LIN {X 0,Y 343.974,Z 466.655,A -85,B 0,C 180,E1 15502.924,E2 15502.924} C_VEL
LIN {X 0,Y 341.205,Z 461.554,A -85,B 0,C 180,E1 15499.694,E2 15499.694} C_VEL
LIN {X 0,Y 339.187,Z 457.553,A -85,B 0,C 180,E1 15496.615,E2 15496.615} C_VEL
LIN {X 0,Y 338.279,Z 456.355,A -85,B 0,C 180,E1 15495.252,E2 15495.252} C_VEL
LIN {X 0,Y 336.252,Z 451.923,A -85,B 0,C 180,E1 15489.413,E2 15489.413} C_VEL
LIN {X 0,Y 335.796,Z 451.415,A -85,B 0,C 180,E1 15484.054,E2 15484.054} C_VEL
LIN {X 0,Y 336.908,Z 452.402,A -85,B 0,C 180,E1 15479.66,E2 15479.66} C_VEL
LIN {X 0,Y 340.362,Z 458.036,A -85,B 0,C 180,E1 15473.083,E2 15473.083} C_VEL
LIN {X 0,Y 342.566,Z 462.05,A -85,B 0,C 180,E1 15470.254,E2 15470.254} C_VEL
LIN {X 0,Y 343.564,Z 463.39,A -85,B 0,C 180,E1 15469.266,E2 15469.266} C_VEL
LIN {X 0,Y 346.154,Z 467.623,A -85,B 0,C 180,E1 15466.895,E2 15466.895} C_VEL
LIN {X 0,Y 352.008,Z 475.085,A -85,B 0,C 180,E1 15463.838,E2 15463.838} C_VEL
LIN {X 0,Y 358.537,Z 483.415,A -85,B 0,C 180,E1 15460.957,E2 15460.957} C_VEL
LIN {X 0,Y 366.447,Z 494.283,A -85,B 0,C 180,E1 15457.924,E2 15457.924} C_VEL
LIN {X 0,Y 375.438,Z 507.505,A -85,B 0,C 180,E1 15454.906,E2 15454.906} C_VEL
LIN {X 0,Y 384.953,Z 522.741,A -85,B 0,C 180,E1 15452.064,E2 15452.064} C_VEL
LIN {X 0,Y 386.963,Z 526.463,A -85,B 0,C 180,E1 15451.489,E2 15451.489} C_VEL
LIN {X 0,Y 374.82,Z 720.746,A -85,B 0,C 180,E1 15447.413,E2 15447.413} C_VEL
LIN {X 0,Y 369.926,Z 797.825,A -85,B 0,C 180,E1 15445.731,E2 15445.731} C_VEL
LIN {X 0,Y 367.045,Z 821.363,A -85,B 0,C 180,E1 15445.019,E2 15445.019} C_VEL
LIN {X 0,Y 363.025,Z 845.088,A -85,B 0,C 180,E1 15444.072,E2 15444.072} C_VEL
LIN {X 0,Y 358.533,Z 867.366,A -85,B 0,C 180,E1 15442.901,E2 15442.901} C_VEL
LIN {X 0,Y 353.441,Z 888.781,A -85,B 0,C 180,E1 15441.463,E2 15441.463} C_VEL
LIN {X 0,Y 347.685,Z 910.726,A -85,B 0,C 180,E1 15439.648,E2 15439.648} C_VEL
LIN {X 0,Y 341.955,Z 930.881,A -85,B 0,C 180,E1 15437.632,E2 15437.632} C_VEL
LIN {X 0,Y 335.907,Z 950.699,A -85,B 0,C 180,E1 15435.229,E2 15435.229} C_VEL
LIN {X 0,Y 329.81,Z 970.146,A -85,B 0,C 180,E1 15432.419,E2 15432.419} C_VEL
LIN {X 0,Y 324.313,Z 987.655,A -85,B 0,C 180,E1 15429.428,E2 15429.428} C_VEL
LIN {X 0,Y 319.205,Z 1004.098,A -85,B 0,C 180,E1 15426.078,E2 15426.078} C_VEL
LIN {X 0,Y 314.594,Z 1019.874,A -85,B 0,C 180,E1 15422.285,E2 15422.285} C_VEL
LIN {X 0,Y 311.178,Z 1032.9,A -85,B 0,C 180,E1 15418.605,E2 15418.605} C_VEL
LIN {X 0,Y 308.521,Z 1044.406,A -85,B 0,C 180,E1 15414.713,E2 15414.713} C_VEL
LIN {X 0,Y 306.649,Z 1054.589,A -85,B 0,C 180,E1 15410.619,E2 15410.619} C_VEL
LIN {X 0,Y 305.659,Z 1062.099,A -85,B 0,C 180,E1 15406.926,E2 15406.926} C_VEL
LIN {X 0,Y 305.155,Z 1068.715,A -85,B 0,C 180,E1 15402.874,E2 15402.874} C_VEL
LIN {X 0,Y 305.04,Z 1073.096,A -85,B 0,C 180,E1 15399.242,E2 15399.242} C_VEL
LIN {X 0,Y 305.141,Z 1075.999,A -85,B 0,C 180,E1 15395.83,E2 15395.83} C_VEL
LIN {X 0,Y 305.246,Z 1077.669,A -85,B 0,C 180,E1 15392.065,E2 15392.065} C_VEL
LIN {X 0,Y 305.248,Z 1077.813,A -85,B 0,C 180,E1 15388.874,E2 15388.874} C_VEL
LIN {X 0,Y 305.192,Z 1076.833,A -85,B 0,C 180,E1 15385.679,E2 15385.679} C_VEL
LIN {X 0,Y 305.078,Z 1074.266,A -85,B 0,C 180,E1 15381.898,E2 15381.898} C_VEL
LIN {X 0,Y 305.105,Z 1069.978,A -85,B 0,C 180,E1 15378.085,E2 15378.085} C_VEL
LIN {X 0,Y 305.427,Z 1064.526,A -85,B 0,C 180,E1 15374.428,E2 15374.428} C_VEL
LIN {X 0,Y 306.341,Z 1056.686,A -85,B 0,C 180,E1 15370.356,E2 15370.356} C_VEL
LIN {X 0,Y 307.902,Z 1047.568,A -85,B 0,C 180,E1 15366.458,E2 15366.458} C_VEL
LIN {X 0,Y 310.287,Z 1036.485,A -85,B 0,C 180,E1 15362.561,E2 15362.561} C_VEL
LIN {X 0,Y 313.609,Z 1023.525,A -85,B 0,C 180,E1 15358.689,E2 15358.689} C_VEL
LIN {X 0,Y 317.476,Z 1009.897,A -85,B 0,C 180,E1 15355.246,E2 15355.246} C_VEL
LIN {X 0,Y 322.515,Z 993.292,A -85,B 0,C 180,E1 15351.681,E2 15351.681} C_VEL
LIN {X 0,Y 327.889,Z 976.235,A -85,B 0,C 180,E1 15348.569,E2 15348.569} C_VEL
LIN {X 0,Y 333.337,Z 958.875,A -85,B 0,C 180,E1 15345.901,E2 15345.901} C_VEL
LIN {X 0,Y 339.647,Z 938.285,A -85,B 0,C 180,E1 15343.231,E2 15343.231} C_VEL
LIN {X 0,Y 345.607,Z 918.087,A -85,B 0,C 180,E1 15341.05,E2 15341.05} C_VEL
LIN {X 0,Y 351.134,Z 897.689,A -85,B 0,C 180,E1 15339.238,E2 15339.238} C_VEL
LIN {X 0,Y 356.626,Z 875.444,A -85,B 0,C 180,E1 15337.623,E2 15337.623} C_VEL
LIN {X 0,Y 361.328,Z 853.913,A -85,B 0,C 180,E1 15336.365,E2 15336.365} C_VEL
LIN {X 0,Y 365.391,Z 831.587,A -85,B 0,C 180,E1 15335.367,E2 15335.367} C_VEL
LIN {X 0,Y 368.882,Z 806.789,A -85,B 0,C 180,E1 15334.53,E2 15334.53} C_VEL
LIN {X 0,Y 370.981,Z 782.961,A -85,B 0,C 180,E1 15333.928,E2 15333.928} C_VEL
LIN {X 0,Y 383.67,Z 577.593,A -85,B 0,C 180,E1 15329.572,E2 15329.572} C_VEL
LIN {X 0,Y 386.794,Z 526.022,A -85,B 0,C 180,E1 15328.485,E2 15328.485} C_VEL
LIN {X 0,Y 378.081,Z 511.736,A -85,B 0,C 180,E1 15325.955,E2 15325.955} C_VEL
LIN {X 0,Y 370.52,Z 500.263,A -85,B 0,C 180,E1 15323.539,E2 15323.539} C_VEL
LIN {X 0,Y 361.938,Z 488.016,A -85,B 0,C 180,E1 15320.454,E2 15320.454} C_VEL
LIN {X 0,Y 354.015,Z 477.663,A -85,B 0,C 180,E1 15317.166,E2 15317.166} C_VEL
LIN {X 0,Y 349.793,Z 472.376,A -85,B 0,C 180,E1 15315.161,E2 15315.161} C_VEL
LIN {X 0,Y 345.844,Z 467.344,A -85,B 0,C 180,E1 15313.032,E2 15313.032} C_VEL
LIN {X 0,Y 342.959,Z 462.497,A -85,B 0,C 180,E1 15310.243,E2 15310.243} C_VEL
LIN {X 0,Y 340.424,Z 458.382,A -85,B 0,C 180,E1 15307.255,E2 15307.255} C_VEL
LIN {X 0,Y 339.834,Z 457.343,A -85,B 0,C 180,E1 15306.419,E2 15306.419} C_VEL
LIN {X 0,Y 336.702,Z 452.103,A -85,B 0,C 180,E1 15300.17,E2 15300.17} C_VEL
LIN {X 0,Y 335.523,Z 451.26,A -85,B 0,C 180,E1 15294.87,E2 15294.87} C_VEL
LIN {X 0,Y 336.345,Z 451.99,A -85,B 0,C 180,E1 15289.898,E2 15289.898} C_VEL
LIN {X 0,Y 339.121,Z 457.459,A -85,B 0,C 180,E1 15283.205,E2 15283.205} C_VEL
LIN {X 0,Y 341.044,Z 461.387,A -85,B 0,C 180,E1 15280.238,E2 15280.238} C_VEL
LIN {X 0,Y 341.808,Z 462.804,A -85,B 0,C 180,E1 15279.27,E2 15279.27} C_VEL
LIN {X 0,Y 344.202,Z 467.421,A -85,B 0,C 180,E1 15276.548,E2 15276.548} C_VEL
LIN {X 0,Y 348.739,Z 473.746,A -85,B 0,C 180,E1 15273.844,E2 15273.844} C_VEL
LIN {X 0,Y 351.856,Z 477.832,A -85,B 0,C 180,E1 15272.314,E2 15272.314} C_VEL
LIN {X 0,Y 358.049,Z 486.342,A -85,B 0,C 180,E1 15269.592,E2 15269.592} C_VEL
LIN {X 0,Y 364.787,Z 496.023,A -85,B 0,C 180,E1 15266.994,E2 15266.994} C_VEL
LIN {X 0,Y 372.893,Z 508.428,A -85,B 0,C 180,E1 15264.229,E2 15264.229} C_VEL
LIN {X 0,Y 381.885,Z 523.465,A -85,B 0,C 180,E1 15261.502,E2 15261.502} C_VEL
LIN {X 0,Y 381.997,Z 527.297,A -85,B 0,C 180,E1 15261.356,E2 15261.356} C_VEL
LIN {X 0,Y 370.72,Z 754.722,A -85,B 0,C 180,E1 15257.08,E2 15257.08} C_VEL
LIN {X 0,Y 368.846,Z 775.36,A -85,B 0,C 180,E1 15256.438,E2 15256.438} C_VEL
LIN {X 0,Y 366.004,Z 796.186,A -85,B 0,C 180,E1 15255.536,E2 15255.536} C_VEL
LIN {X 0,Y 362.593,Z 815.194,A -85,B 0,C 180,E1 15254.46,E2 15254.46} C_VEL
LIN {X 0,Y 358.372,Z 833.832,A -85,B 0,C 180,E1 15253.122,E2 15253.122} C_VEL
LIN {X 0,Y 353.575,Z 851.659,A -85,B 0,C 180,E1 15251.54,E2 15251.54} C_VEL
LIN {X 0,Y 348.388,Z 868.504,A -85,B 0,C 180,E1 15249.722,E2 15249.722} C_VEL
LIN {X 0,Y 342.699,Z 884.886,A -85,B 0,C 180,E1 15247.574,E2 15247.574} C_VEL
LIN {X 0,Y 336.914,Z 899.931,A -85,B 0,C 180,E1 15245.151,E2 15245.151} C_VEL
LIN {X 0,Y 331.245,Z 913.564,A -85,B 0,C 180,E1 15242.5,E2 15242.5} C_VEL
LIN {X 0,Y 325.925,Z 925.847,A -85,B 0,C 180,E1 15239.598,E2 15239.598} C_VEL
LIN {X 0,Y 320.751,Z 937.321,A -85,B 0,C 180,E1 15236.273,E2 15236.273} C_VEL
LIN {X 0,Y 316.26,Z 947.14,A -85,B 0,C 180,E1 15232.688,E2 15232.688} C_VEL
LIN {X 0,Y 312.692,Z 955.048,A -85,B 0,C 180,E1 15229.036,E2 15229.036} C_VEL
LIN {X 0,Y 309.839,Z 961.81,A -85,B 0,C 180,E1 15224.961,E2 15224.961} C_VEL
LIN {X 0,Y 308.026,Z 966.572,A -85,B 0,C 180,E1 15221.041,E2 15221.041} C_VEL
LIN {X 0,Y 306.914,Z 969.924,A -85,B 0,C 180,E1 15216.923,E2 15216.923} C_VEL
LIN {X 0,Y 306.384,Z 971.643,A -85,B 0,C 180,E1 15212.806,E2 15212.806} C_VEL
LIN {X 0,Y 306.299,Z 971.927,A -85,B 0,C 180,E1 15208.878,E2 15208.878} C_VEL
LIN {X 0,Y 306.619,Z 970.836,A -85,B 0,C 180,E1 15204.761,E2 15204.761} C_VEL
LIN {X 0,Y 307.474,Z 968.249,A -85,B 0,C 180,E1 15200.643,E2 15200.643} C_VEL
LIN {X 0,Y 309.005,Z 963.97,A -85,B 0,C 180,E1 15196.528,E2 15196.528} C_VEL
LIN {X 0,Y 311.364,Z 958.227,A -85,B 0,C 180,E1 15192.624,E2 15192.624} C_VEL
LIN {X 0,Y 314.49,Z 951.056,A -85,B 0,C 180,E1 15188.907,E2 15188.907} C_VEL
LIN {X 0,Y 314.88,Z 948.415,A -85,B 0,C 180,E1 15187.58,E2 15187.58} C_VEL
LIN {X 0,Y 313.132,Z 941.752,A -85,B 0,C 180,E1 15184.124,E2 15184.124} C_VEL
LIN {X 0,Y 313.889,Z 938.359,A -85,B 0,C 180,E1 15182.856,E2 15182.856} C_VEL
LIN {X 0,Y 319.273,Z 926.988,A -85,B 0,C 180,E1 15179.514,E2 15179.514} C_VEL
LIN {X 0,Y 324.842,Z 914.675,A -85,B 0,C 180,E1 15176.567,E2 15176.567} C_VEL
LIN {X 0,Y 331.139,Z 900.064,A -85,B 0,C 180,E1 15173.714,E2 15173.714} C_VEL
LIN {X 0,Y 336.987,Z 885.362,A -85,B 0,C 180,E1 15171.349,E2 15171.349} C_VEL
LIN {X 0,Y 342.841,Z 869.118,A -85,B 0,C 180,E1 15169.211,E2 15169.211} C_VEL
LIN {X 0,Y 348.074,Z 852.672,A -85,B 0,C 180,E1 15167.43,E2 15167.43} C_VEL
LIN {X 0,Y 353.045,Z 834.833,A -85,B 0,C 180,E1 15165.837,E2 15165.837} C_VEL
LIN {X 0,Y 357.415,Z 816.203,A -85,B 0,C 180,E1 15164.491,E2 15164.491} C_VEL
LIN {X 0,Y 361.075,Z 796.506,A -85,B 0,C 180,E1 15163.373,E2 15163.373} C_VEL
LIN {X 0,Y 364.016,Z 775.499,A -85,B 0,C 180,E1 15162.468,E2 15162.468} C_VEL
LIN {X 0,Y 365.927,Z 754.887,A -85,B 0,C 180,E1 15161.83,E2 15161.83} C_VEL
LIN {X 0,Y 377.655,Z 527.845,A -85,B 0,C 180,E1 15157.513,E2 15157.513} C_VEL
LIN {X 0,Y 369.147,Z 513.555,A -85,B 0,C 180,E1 15154.809,E2 15154.809} C_VEL
LIN {X 0,Y 361.207,Z 501.26,A -85,B 0,C 180,E1 15151.965,E2 15151.965} C_VEL
LIN {X 0,Y 354.549,Z 491.6,A -85,B 0,C 180,E1 15149.248,E2 15149.248} C_VEL
LIN {X 0,Y 348.202,Z 482.708,A -85,B 0,C 180,E1 15146.245,E2 15146.245} C_VEL
LIN {X 0,Y 341.714,Z 474.041,A -85,B 0,C 180,E1 15142.539,E2 15142.539} C_VEL
LIN {X 0,Y 338.064,Z 469.215,A -85,B 0,C 180,E1 15139.975,E2 15139.975} C_VEL
LIN {X 0,Y 335.758,Z 465.827,A -85,B 0,C 180,E1 15137.326,E2 15137.326} C_VEL
LIN {X 0,Y 335.009,Z 463.83,A -85,B 0,C 180,E1 15135.76,E2 15135.76} C_VEL
LIN {X 0,Y 332.7,Z 459.081,A -85,B 0,C 180,E1 15129.34,E2 15129.34} C_VEL
LIN {X 0,Y 332.274,Z 458.602,A -85,B 0,C 180,E1 15123.969,E2 15123.969} C_VEL
LIN {X 0,Y 333.405,Z 459.621,A -85,B 0,C 180,E1 15119.657,E2 15119.657} C_VEL
LIN {X 0,Y 336.734,Z 465.24,A -85,B 0,C 180,E1 15113.179,E2 15113.179} C_VEL
LIN {X 0,Y 338.642,Z 468.549,A -85,B 0,C 180,E1 15110.998,E2 15110.998} C_VEL
LIN {X 0,Y 340.885,Z 470.946,A -85,B 0,C 180,E1 15109.437,E2 15109.437} C_VEL
LIN {X 0,Y 345.367,Z 476.472,A -85,B 0,C 180,E1 15106.694,E2 15106.694} C_VEL
LIN {X 0,Y 350.089,Z 482.514,A -85,B 0,C 180,E1 15104.215,E2 15104.215} C_VEL
LIN {X 0,Y 356.404,Z 490.785,A -85,B 0,C 180,E1 15101.349,E2 15101.349} C_VEL
LIN {X 0,Y 363.89,Z 501.241,A -85,B 0,C 180,E1 15098.396,E2 15098.396} C_VEL
LIN {X 0,Y 372.816,Z 514.664,A -85,B 0,C 180,E1 15095.311,E2 15095.311} C_VEL
LIN {X 0,Y 381.781,Z 529.373,A -85,B 0,C 180,E1 15092.553,E2 15092.553} C_VEL
LIN {X 0,Y 382.259,Z 530.611,A -85,B 0,C 180,E1 15092.4,E2 15092.4} C_VEL
LIN {X 0,Y 369.496,Z 728.067,A -85,B 0,C 180,E1 15088.238,E2 15088.238} C_VEL
LIN {X 0,Y 364.921,Z 797.295,A -85,B 0,C 180,E1 15086.716,E2 15086.716} C_VEL
LIN {X 0,Y 361.961,Z 820.778,A -85,B 0,C 180,E1 15086.002,E2 15086.002} C_VEL
LIN {X 0,Y 357.789,Z 844.591,A -85,B 0,C 180,E1 15085.049,E2 15085.049} C_VEL
LIN {X 0,Y 353.133,Z 866.83,A -85,B 0,C 180,E1 15083.875,E2 15083.875} C_VEL
LIN {X 0,Y 347.716,Z 888.76,A -85,B 0,C 180,E1 15082.392,E2 15082.392} C_VEL
LIN {X 0,Y 341.748,Z 910.507,A -85,B 0,C 180,E1 15080.57,E2 15080.57} C_VEL
LIN {X 0,Y 335.713,Z 930.832,A -85,B 0,C 180,E1 15078.503,E2 15078.503} C_VEL
LIN {X 0,Y 329.57,Z 950.06,A -85,B 0,C 180,E1 15076.133,E2 15076.133} C_VEL
LIN {X 0,Y 323.088,Z 969.683,A -85,B 0,C 180,E1 15073.246,E2 15073.246} C_VEL
LIN {X 0,Y 317.223,Z 987.432,A -85,B 0,C 180,E1 15070.134,E2 15070.134} C_VEL
LIN {X 0,Y 312.017,Z 1003.337,A -85,B 0,C 180,E1 15066.816,E2 15066.816} C_VEL
LIN {X 0,Y 307.367,Z 1018.332,A -85,B 0,C 180,E1 15063.128,E2 15063.128} C_VEL
LIN {X 0,Y 303.597,Z 1031.821,A -85,B 0,C 180,E1 15059.222,E2 15059.222} C_VEL
LIN {X 0,Y 300.754,Z 1043.422,A -85,B 0,C 180,E1 15055.185,E2 15055.185} C_VEL
LIN {X 0,Y 298.775,Z 1053.528,A -85,B 0,C 180,E1 15050.982,E2 15050.982} C_VEL
LIN {X 0,Y 297.731,Z 1061.003,A -85,B 0,C 180,E1 15047.189,E2 15047.189} C_VEL
LIN {X 0,Y 297.219,Z 1067.547,A -85,B 0,C 180,E1 15043.026,E2 15043.026} C_VEL
LIN {X 0,Y 297.115,Z 1071.696,A -85,B 0,C 180,E1 15039.491,E2 15039.491} C_VEL
LIN {X 0,Y 297.245,Z 1074.62,A -85,B 0,C 180,E1 15035.985,E2 15035.985} C_VEL
LIN {X 0,Y 297.358,Z 1076.302,A -85,B 0,C 180,E1 15032.12,E2 15032.12} C_VEL
LIN {X 0,Y 297.365,Z 1076.447,A -85,B 0,C 180,E1 15028.844,E2 15028.844} C_VEL
LIN {X 0,Y 297.294,Z 1075.458,A -85,B 0,C 180,E1 15025.563,E2 15025.563} C_VEL
LIN {X 0,Y 297.164,Z 1073.048,A -85,B 0,C 180,E1 15021.876,E2 15021.876} C_VEL
LIN {X 0,Y 297.174,Z 1068.811,A -85,B 0,C 180,E1 15017.959,E2 15017.959} C_VEL
LIN {X 0,Y 297.499,Z 1063.392,A -85,B 0,C 180,E1 15014.203,E2 15014.203} C_VEL
LIN {X 0,Y 298.443,Z 1055.623,A -85,B 0,C 180,E1 15010.018,E2 15010.018} C_VEL
LIN {X 0,Y 299.989,Z 1047.02,A -85,B 0,C 180,E1 15006.216,E2 15006.216} C_VEL
LIN {X 0,Y 302.462,Z 1036.135,A -85,B 0,C 180,E1 15002.218,E2 15002.218} C_VEL
LIN {X 0,Y 305.92,Z 1023.385,A -85,B 0,C 180,E1 14998.25,E2 14998.25} C_VEL
LIN {X 0,Y 310.195,Z 1009.083,A -85,B 0,C 180,E1 14994.535,E2 14994.535} C_VEL
LIN {X 0,Y 315.486,Z 992.578,A -85,B 0,C 180,E1 14990.899,E2 14990.899} C_VEL
LIN {X 0,Y 321.139,Z 975.638,A -85,B 0,C 180,E1 14987.738,E2 14987.738} C_VEL
LIN {X 0,Y 327.07,Z 957.6,A -85,B 0,C 180,E1 14984.923,E2 14984.923} C_VEL
LIN {X 0,Y 333.629,Z 937.172,A -85,B 0,C 180,E1 14982.248,E2 14982.248} C_VEL
LIN {X 0,Y 339.766,Z 917.287,A -85,B 0,C 180,E1 14980.081,E2 14980.081} C_VEL
LIN {X 0,Y 345.491,Z 896.992,A -85,B 0,C 180,E1 14978.266,E2 14978.266} C_VEL
LIN {X 0,Y 351.284,Z 874.352,A -85,B 0,C 180,E1 14976.615,E2 14976.615} C_VEL
LIN {X 0,Y 356.178,Z 852.663,A -85,B 0,C 180,E1 14975.35,E2 14975.35} C_VEL
LIN {X 0,Y 360.379,Z 830.197,A -85,B 0,C 180,E1 14974.352,E2 14974.352} C_VEL
LIN {X 0,Y 363.929,Z 805.476,A -85,B 0,C 180,E1 14973.525,E2 14973.525} C_VEL
LIN {X 0,Y 366.084,Z 781.261,A -85,B 0,C 180,E1 14972.916,E2 14972.916} C_VEL
LIN {X 0,Y 379.142,Z 577.108,A -85,B 0,C 180,E1 14968.57,E2 14968.57} C_VEL
LIN {X 0,Y 382.085,Z 530.038,A -85,B 0,C 180,E1 14967.571,E2 14967.571} C_VEL
LIN {X 0,Y 374.108,Z 516.865,A -85,B 0,C 180,E1 14965.147,E2 14965.147} C_VEL
LIN {X 0,Y 367.26,Z 506.362,A -85,B 0,C 180,E1 14962.869,E2 14962.869} C_VEL
LIN {X 0,Y 359.461,Z 494.995,A -85,B 0,C 180,E1 14959.964,E2 14959.964} C_VEL
LIN {X 0,Y 351.97,Z 484.981,A -85,B 0,C 180,E1 14956.758,E2 14956.758} C_VEL
LIN {X 0,Y 347.835,Z 479.71,A -85,B 0,C 180,E1 14954.737,E2 14954.737} C_VEL
LIN {X 0,Y 343.952,Z 474.731,A -85,B 0,C 180,E1 14952.592,E2 14952.592} C_VEL
LIN {X 0,Y 339.747,Z 469.644,A -85,B 0,C 180,E1 14949.913,E2 14949.913} C_VEL
LIN {X 0,Y 336.992,Z 466.115,A -85,B 0,C 180,E1 14947.501,E2 14947.501} C_VEL
LIN {X 0,Y 336.247,Z 464.471,A -85,B 0,C 180,E1 14946.316,E2 14946.316} C_VEL
LIN {X 0,Y 333.205,Z 459.312,A -85,B 0,C 180,E1 14940.171,E2 14940.171} C_VEL
LIN {X 0,Y 331.998,Z 458.438,A -85,B 0,C 180,E1 14934.989,E2 14934.989} C_VEL
LIN {X 0,Y 332.745,Z 459.126,A -85,B 0,C 180,E1 14929.963,E2 14929.963} C_VEL
LIN {X 0,Y 335.313,Z 464.463,A -85,B 0,C 180,E1 14923.365,E2 14923.365} C_VEL
LIN {X 0,Y 337.249,Z 468.357,A -85,B 0,C 180,E1 14920.426,E2 14920.426} C_VEL
LIN {X 0,Y 338.525,Z 470.119,A -85,B 0,C 180,E1 14919.422,E2 14919.422} C_VEL
LIN {X 0,Y 342.714,Z 475.552,A -85,B 0,C 180,E1 14916.623,E2 14916.623} C_VEL
LIN {X 0,Y 348.932,Z 483.649,A -85,B 0,C 180,E1 14913.217,E2 14913.217} C_VEL
LIN {X 0,Y 356.118,Z 493.943,A -85,B 0,C 180,E1 14909.922,E2 14909.922} C_VEL
LIN {X 0,Y 362.767,Z 503.721,A -85,B 0,C 180,E1 14907.301,E2 14907.301} C_VEL
LIN {X 0,Y 370.116,Z 515.249,A -85,B 0,C 180,E1 14904.729,E2 14904.729} C_VEL
LIN {X 0,Y 377.635,Z 528.076,A -85,B 0,C 180,E1 14902.361,E2 14902.361} C_VEL
LIN {X 0,Y 365.808,Z 755.43,A -85,B 0,C 180,E1 14898.056,E2 14898.056} C_VEL
LIN {X 0,Y 363.855,Z 776.124,A -85,B 0,C 180,E1 14897.409,E2 14897.409} C_VEL
LIN {X 0,Y 360.866,Z 797.225,A -85,B 0,C 180,E1 14896.489,E2 14896.489} C_VEL
LIN {X 0,Y 357.174,Z 816.9,A -85,B 0,C 180,E1 14895.36,E2 14895.36} C_VEL
LIN {X 0,Y 352.734,Z 835.787,A -85,B 0,C 180,E1 14893.986,E2 14893.986} C_VEL
LIN {X 0,Y 347.747,Z 853.498,A -85,B 0,C 180,E1 14892.385,E2 14892.385} C_VEL
LIN {X 0,Y 341.876,Z 871.62,A -85,B 0,C 180,E1 14890.377,E2 14890.377} C_VEL
LIN {X 0,Y 336.095,Z 887.515,A -85,B 0,C 180,E1 14888.228,E2 14888.228} C_VEL
LIN {X 0,Y 330.137,Z 902.402,A -85,B 0,C 180,E1 14885.77,E2 14885.77} C_VEL
LIN {X 0,Y 324.277,Z 915.819,A -85,B 0,C 180,E1 14883.076,E2 14883.076} C_VEL
LIN {X 0,Y 318.428,Z 928.63,A -85,B 0,C 180,E1 14879.929,E2 14879.929} C_VEL
LIN {X 0,Y 313.346,Z 939.384,A -85,B 0,C 180,E1 14876.688,E2 14876.688} C_VEL
LIN {X 0,Y 308.76,Z 949.009,A -85,B 0,C 180,E1 14873.069,E2 14873.069} C_VEL
LIN {X 0,Y 304.958,Z 957.012,A -85,B 0,C 180,E1 14869.219,E2 14869.219} C_VEL
LIN {X 0,Y 302.19,Z 963.193,A -85,B 0,C 180,E1 14865.349,E2 14865.349} C_VEL
LIN {X 0,Y 300.19,Z 968.121,A -85,B 0,C 180,E1 14861.139,E2 14861.139} C_VEL
LIN {X 0,Y 299.077,Z 971.293,A -85,B 0,C 180,E1 14857.106,E2 14857.106} C_VEL
LIN {X 0,Y 298.507,Z 973.01,A -85,B 0,C 180,E1 14852.88,E2 14852.88} C_VEL
LIN {X 0,Y 298.418,Z 973.292,A -85,B 0,C 180,E1 14848.848,E2 14848.848} C_VEL
LIN {X 0,Y 298.761,Z 972.203,A -85,B 0,C 180,E1 14844.623,E2 14844.623} C_VEL
LIN {X 0,Y 299.674,Z 969.621,A -85,B 0,C 180,E1 14840.397,E2 14840.397} C_VEL
LIN {X 0,Y 301.307,Z 965.347,A -85,B 0,C 180,E1 14836.177,E2 14836.177} C_VEL
LIN {X 0,Y 303.804,Z 959.612,A -85,B 0,C 180,E1 14832.177,E2 14832.177} C_VEL
LIN {X 0,Y 307.259,Z 952.126,A -85,B 0,C 180,E1 14828.224,E2 14828.224} C_VEL
LIN {X 0,Y 311.57,Z 943.154,A -85,B 0,C 180,E1 14824.531,E2 14824.531} C_VEL
LIN {X 0,Y 313.889,Z 938.359,A -85,B 0,C 180,E1 14822.856,E2 14822.856} C_VEL
LIN {X 0,Y 314.744,Z 934.836,A -85,B 0,C 180,E1 14821.61,E2 14821.61} C_VEL
LIN {X 0,Y 314.325,Z 926.159,A -85,B 0,C 180,E1 14818.307,E2 14818.307} C_VEL
LIN {X 0,Y 315.576,Z 921.965,A -85,B 0,C 180,E1 14817.129,E2 14817.129} C_VEL
LIN {X 0,Y 321.754,Z 908.546,A -85,B 0,C 180,E1 14814.201,E2 14814.201} C_VEL
LIN {X 0,Y 328.22,Z 893.534,A -85,B 0,C 180,E1 14811.528,E2 14811.528} C_VEL
LIN {X 0,Y 334.217,Z 878.324,A -85,B 0,C 180,E1 14809.294,E2 14809.294} C_VEL
LIN {X 0,Y 340.217,Z 861.159,A -85,B 0,C 180,E1 14807.243,E2 14807.243} C_VEL
LIN {X 0,Y 345.516,Z 843.84,A -85,B 0,C 180,E1 14805.548,E2 14805.548} C_VEL
LIN {X 0,Y 350.34,Z 825.554,A -85,B 0,C 180,E1 14804.087,E2 14804.087} C_VEL
LIN {X 0,Y 354.296,Z 807.283,A -85,B 0,C 180,E1 14802.917,E2 14802.917} C_VEL
LIN {X 0,Y 357.665,Z 787.369,A -85,B 0,C 180,E1 14801.919,E2 14801.919} C_VEL
LIN {X 0,Y 360.171,Z 766.869,A -85,B 0,C 180,E1 14801.148,E2 14801.148} C_VEL
LIN {X 0,Y 361.729,Z 745.715,A -85,B 0,C 180,E1 14800.6,E2 14800.6} C_VEL
LIN {X 0,Y 373.246,Z 531.923,A -85,B 0,C 180,E1 14796.552,E2 14796.552} C_VEL
LIN {X 0,Y 364.866,Z 517.88,A -85,B 0,C 180,E1 14793.753,E2 14793.753} C_VEL
LIN {X 0,Y 357.885,Z 506.971,A -85,B 0,C 180,E1 14791.122,E2 14791.122} C_VEL
LIN {X 0,Y 351.891,Z 498.044,A -85,B 0,C 180,E1 14788.56,E2 14788.56} C_VEL
LIN {X 0,Y 346.048,Z 489.737,A -85,B 0,C 180,E1 14785.684,E2 14785.684} C_VEL
LIN {X 0,Y 340.123,Z 481.605,A -85,B 0,C 180,E1 14782.179,E2 14782.179} C_VEL
LIN {X 0,Y 335.951,Z 476.14,A -85,B 0,C 180,E1 14779.11,E2 14779.11} C_VEL
LIN {X 0,Y 332.24,Z 471.267,A -85,B 0,C 180,E1 14775.536,E2 14775.536} C_VEL
LIN {X 0,Y 329.308,Z 466.828,A -85,B 0,C 180,E1 14770.32,E2 14770.32} C_VEL
LIN {X 0,Y 328.869,Z 465.945,A -85,B 0,C 180,E1 14767.864,E2 14767.864} C_VEL
LIN {X 0,Y 329.092,Z 466.025,A -85,B 0,C 180,E1 14762.264,E2 14762.264} C_VEL
LIN {X 0,Y 329.974,Z 467.019,A -85,B 0,C 180,E1 14759.397,E2 14759.397} C_VEL
LIN {X 0,Y 334.712,Z 472.907,A -85,B 0,C 180,E1 14753.396,E2 14753.396} C_VEL
LIN {X 0,Y 339.413,Z 478.686,A -85,B 0,C 180,E1 14749.712,E2 14749.712} C_VEL
LIN {X 0,Y 343.638,Z 483.995,A -85,B 0,C 180,E1 14747.054,E2 14747.054} C_VEL
LIN {X 0,Y 348.185,Z 489.944,A -85,B 0,C 180,E1 14744.596,E2 14744.596} C_VEL
LIN {X 0,Y 354.208,Z 498.011,A -85,B 0,C 180,E1 14741.783,E2 14741.783} C_VEL
LIN {X 0,Y 361.449,Z 508.343,A -85,B 0,C 180,E1 14738.839,E2 14738.839} C_VEL
LIN {X 0,Y 370.105,Z 521.665,A -85,B 0,C 180,E1 14735.756,E2 14735.756} C_VEL
LIN {X 0,Y 377.68,Z 534.326,A -85,B 0,C 180,E1 14733.341,E2 14733.341} C_VEL
LIN {X 0,Y 364.39,Z 733.159,A -85,B 0,C 180,E1 14729.135,E2 14729.135} C_VEL
LIN {X 0,Y 360.038,Z 796.661,A -85,B 0,C 180,E1 14727.73,E2 14727.73} C_VEL
LIN {X 0,Y 356.981,Z 820.227,A -85,B 0,C 180,E1 14727.012,E2 14727.012} C_VEL
LIN {X 0,Y 352.754,Z 843.661,A -85,B 0,C 180,E1 14726.075,E2 14726.075} C_VEL
LIN {X 0,Y 348.076,Z 865.368,A -85,B 0,C 180,E1 14724.936,E2 14724.936} C_VEL
LIN {X 0,Y 342.643,Z 886.645,A -85,B 0,C 180,E1 14723.508,E2 14723.508} C_VEL
LIN {X 0,Y 336.42,Z 908.571,A -85,B 0,C 180,E1 14721.686,E2 14721.686} C_VEL
LIN {X 0,Y 330.087,Z 929.157,A -85,B 0,C 180,E1 14719.593,E2 14719.593} C_VEL
LIN {X 0,Y 323.86,Z 947.813,A -85,B 0,C 180,E1 14717.289,E2 14717.289} C_VEL
LIN {X 0,Y 317.12,Z 967.302,A -85,B 0,C 180,E1 14714.424,E2 14714.424} C_VEL
LIN {X 0,Y 311.046,Z 984.829,A -85,B 0,C 180,E1 14711.345,E2 14711.345} C_VEL
LIN {X 0,Y 305.33,Z 1001.246,A -85,B 0,C 180,E1 14707.89,E2 14707.89} C_VEL
LIN {X 0,Y 300.153,Z 1016.986,A -85,B 0,C 180,E1 14703.958,E2 14703.958} C_VEL
LIN {X 0,Y 296.141,Z 1030.423,A -85,B 0,C 180,E1 14699.98,E2 14699.98} C_VEL
LIN {X 0,Y 293.127,Z 1041.904,A -85,B 0,C 180,E1 14695.888,E2 14695.888} C_VEL
LIN {X 0,Y 290.913,Z 1052.47,A -85,B 0,C 180,E1 14691.366,E2 14691.366} C_VEL
LIN {X 0,Y 289.809,Z 1059.911,A -85,B 0,C 180,E1 14687.467,E2 14687.467} C_VEL
LIN {X 0,Y 289.284,Z 1066.38,A -85,B 0,C 180,E1 14683.186,E2 14683.186} C_VEL
LIN {X 0,Y 289.192,Z 1070.494,A -85,B 0,C 180,E1 14679.553,E2 14679.553} C_VEL
LIN {X 0,Y 289.34,Z 1073.514,A -85,B 0,C 180,E1 14675.751,E2 14675.751} C_VEL
LIN {X 0,Y 289.479,Z 1074.966,A -85,B 0,C 180,E1 14671.979,E2 14671.979} C_VEL
LIN {X 0,Y 289.485,Z 1075.054,A -85,B 0,C 180,E1 14668.615,E2 14668.615} C_VEL
LIN {X 0,Y 289.372,Z 1073.908,A -85,B 0,C 180,E1 14665.044,E2 14665.044} C_VEL
LIN {X 0,Y 289.209,Z 1071.08,A -85,B 0,C 180,E1 14661.05,E2 14661.05} C_VEL
LIN {X 0,Y 289.255,Z 1067.139,A -85,B 0,C 180,E1 14657.422,E2 14657.422} C_VEL
LIN {X 0,Y 289.662,Z 1061.325,A -85,B 0,C 180,E1 14653.351,E2 14653.351} C_VEL
LIN {X 0,Y 290.687,Z 1053.721,A -85,B 0,C 180,E1 14649.25,E2 14649.25} C_VEL
LIN {X 0,Y 292.514,Z 1044.553,A -85,B 0,C 180,E1 14645.138,E2 14645.138} C_VEL
LIN {X 0,Y 295.281,Z 1033.396,A -85,B 0,C 180,E1 14641.039,E2 14641.039} C_VEL
LIN {X 0,Y 299.086,Z 1020.351,A -85,B 0,C 180,E1 14636.981,E2 14636.981} C_VEL
LIN {X 0,Y 303.494,Z 1006.686,A -85,B 0,C 180,E1 14633.394,E2 14633.394} C_VEL
LIN {X 0,Y 309.027,Z 990.385,A -85,B 0,C 180,E1 14629.78,E2 14629.78} C_VEL
LIN {X 0,Y 314.921,Z 973.655,A -85,B 0,C 180,E1 14626.64,E2 14626.64} C_VEL
LIN {X 0,Y 321.089,Z 955.805,A -85,B 0,C 180,E1 14623.83,E2 14623.83} C_VEL
LIN {X 0,Y 327.753,Z 935.968,A -85,B 0,C 180,E1 14621.218,E2 14621.218} C_VEL
LIN {X 0,Y 334.159,Z 916.054,A -85,B 0,C 180,E1 14619.038,E2 14619.038} C_VEL
LIN {X 0,Y 339.898,Z 896.488,A -85,B 0,C 180,E1 14617.277,E2 14617.277} C_VEL
LIN {X 0,Y 345.772,Z 874.449,A -85,B 0,C 180,E1 14615.652,E2 14615.652} C_VEL
LIN {X 0,Y 350.647,Z 853.646,A -85,B 0,C 180,E1 14614.425,E2 14614.425} C_VEL
LIN {X 0,Y 355.083,Z 831.103,A -85,B 0,C 180,E1 14613.402,E2 14613.402} C_VEL
LIN {X 0,Y 358.691,Z 807.631,A -85,B 0,C 180,E1 14612.591,E2 14612.591} C_VEL
LIN {X 0,Y 360.959,Z 784.51,A -85,B 0,C 180,E1 14611.989,E2 14611.989} C_VEL
LIN {X 0,Y 374.374,Z 582.053,A -85,B 0,C 180,E1 14607.658,E2 14607.658} C_VEL
LIN {X 0,Y 377.495,Z 534.077,A -85,B 0,C 180,E1 14606.637,E2 14606.637} C_VEL
LIN {X 0,Y 368.44,Z 519.057,A -85,B 0,C 180,E1 14603.722,E2 14603.722} C_VEL
LIN {X 0,Y 359.603,Z 505.746,A -85,B 0,C 180,E1 14600.507,E2 14600.507} C_VEL
LIN {X 0,Y 352.593,Z 495.932,A -85,B 0,C 180,E1 14597.577,E2 14597.577} C_VEL
LIN {X 0,Y 346.508,Z 487.717,A -85,B 0,C 180,E1 14594.624,E2 14594.624} C_VEL
LIN {X 0,Y 342.11,Z 482.12,A -85,B 0,C 180,E1 14592.147,E2 14592.147} C_VEL
LIN {X 0,Y 338.147,Z 477.2,A -85,B 0,C 180,E1 14589.531,E2 14589.531} C_VEL
LIN {X 0,Y 334.065,Z 472.129,A -85,B 0,C 180,E1 14586.185,E2 14586.185} C_VEL
LIN {X 0,Y 329.765,Z 466.613,A -85,B 0,C 180,E1 14580.347,E2 14580.347} C_VEL
LIN {X 0,Y 328.508,Z 465.626,A -85,B 0,C 180,E1 14575.286,E2 14575.286} C_VEL
LIN {X 0,Y 329.143,Z 466.26,A -85,B 0,C 180,E1 14570.028,E2 14570.028} C_VEL
LIN {X 0,Y 330.569,Z 469.617,A -85,B 0,C 180,E1 14566.149,E2 14566.149} C_VEL
LIN {X 0,Y 332.75,Z 471.94,A -85,B 0,C 180,E1 14563.593,E2 14563.593} C_VEL
LIN {X 0,Y 336.09,Z 476.274,A -85,B 0,C 180,E1 14560.537,E2 14560.537} C_VEL
LIN {X 0,Y 341.18,Z 483.221,A -85,B 0,C 180,E1 14556.927,E2 14556.927} C_VEL
LIN {X 0,Y 347.061,Z 491.081,A -85,B 0,C 180,E1 14553.616,E2 14553.616} C_VEL
LIN {X 0,Y 353.848,Z 500.995,A -85,B 0,C 180,E1 14550.41,E2 14550.41} C_VEL
LIN {X 0,Y 360.951,Z 511.682,A -85,B 0,C 180,E1 14547.54,E2 14547.54} C_VEL
LIN {X 0,Y 368.648,Z 524.259,A -85,B 0,C 180,E1 14544.805,E2 14544.805} C_VEL
LIN {X 0,Y 373.199,Z 532.134,A -85,B 0,C 180,E1 14543.328,E2 14543.328} C_VEL
LIN {X 0,Y 361.005,Z 756.112,A -85,B 0,C 180,E1 14539.059,E2 14539.059} C_VEL
LIN {X 0,Y 358.97,Z 776.874,A -85,B 0,C 180,E1 14538.407,E2 14538.407} C_VEL
LIN {X 0,Y 355.829,Z 798.251,A -85,B 0,C 180,E1 14537.469,E2 14537.469} C_VEL
LIN {X 0,Y 352.126,Z 817.386,A -85,B 0,C 180,E1 14536.37,E2 14536.37} C_VEL
LIN {X 0,Y 347.66,Z 835.802,A -85,B 0,C 180,E1 14535.031,E2 14535.031} C_VEL
LIN {X 0,Y 342.566,Z 853.498,A -85,B 0,C 180,E1 14533.442,E2 14533.442} C_VEL
LIN {X 0,Y 336.877,Z 870.721,A -85,B 0,C 180,E1 14531.557,E2 14531.557} C_VEL
LIN {X 0,Y 330.831,Z 886.924,A -85,B 0,C 180,E1 14529.396,E2 14529.396} C_VEL
LIN {X 0,Y 324.575,Z 902.026,A -85,B 0,C 180,E1 14526.921,E2 14526.921} C_VEL
LIN {X 0,Y 318.424,Z 915.724,A -85,B 0,C 180,E1 14524.199,E2 14524.199} C_VEL
LIN {X 0,Y 312.608,Z 928.077,A -85,B 0,C 180,E1 14521.208,E2 14521.208} C_VEL
LIN {X 0,Y 307.18,Z 939.03,A -85,B 0,C 180,E1 14517.951,E2 14517.951} C_VEL
LIN {X 0,Y 302.375,Z 948.569,A -85,B 0,C 180,E1 14514.415,E2 14514.415} C_VEL
LIN {X 0,Y 298.096,Z 957.117,A -85,B 0,C 180,E1 14510.416,E2 14510.416} C_VEL
LIN {X 0,Y 294.933,Z 963.787,A -85,B 0,C 180,E1 14506.343,E2 14506.343} C_VEL
LIN {X 0,Y 292.658,Z 968.973,A -85,B 0,C 180,E1 14502.029,E2 14502.029} C_VEL
LIN {X 0,Y 291.327,Z 972.399,A -85,B 0,C 180,E1 14497.692,E2 14497.692} C_VEL
LIN {X 0,Y 290.671,Z 974.207,A -85,B 0,C 180,E1 14493.55,E2 14493.55} C_VEL
LIN {X 0,Y 290.528,Z 974.696,A -85,B 0,C 180,E1 14489.211,E2 14489.211} C_VEL
LIN {X 0,Y 290.827,Z 973.848,A -85,B 0,C 180,E1 14485.069,E2 14485.069} C_VEL
LIN {X 0,Y 291.696,Z 971.4,A -85,B 0,C 180,E1 14480.729,E2 14480.729} C_VEL
LIN {X 0,Y 293.318,Z 967.376,A -85,B 0,C 180,E1 14476.396,E2 14476.396} C_VEL
LIN {X 0,Y 295.976,Z 961.614,A -85,B 0,C 180,E1 14472.096,E2 14472.096} C_VEL
LIN {X 0,Y 299.519,Z 954.337,A -85,B 0,C 180,E1 14468.045,E2 14468.045} C_VEL
LIN {X 0,Y 303.952,Z 945.585,A -85,B 0,C 180,E1 14464.264,E2 14464.264} C_VEL
LIN {X 0,Y 309.075,Z 935.299,A -85,B 0,C 180,E1 14460.759,E2 14460.759} C_VEL
LIN {X 0,Y 314.787,Z 923.595,A -85,B 0,C 180,E1 14457.534,E2 14457.534} C_VEL
LIN {X 0,Y 315.576,Z 921.965,A -85,B 0,C 180,E1 14457.129,E2 14457.129} C_VEL
LIN {X 0,Y 316.903,Z 917.709,A -85,B 0,C 180,E1 14455.976,E2 14455.976} C_VEL
LIN {X 0,Y 317.547,Z 906.996,A -85,B 0,C 180,E1 14452.904,E2 14452.904} C_VEL
LIN {X 0,Y 319.035,Z 902.075,A -85,B 0,C 180,E1 14451.858,E2 14451.858} C_VEL
LIN {X 0,Y 325.552,Z 886.801,A -85,B 0,C 180,E1 14449.374,E2 14449.374} C_VEL
LIN {X 0,Y 331.862,Z 870.461,A -85,B 0,C 180,E1 14447.203,E2 14447.203} C_VEL
LIN {X 0,Y 337.733,Z 853.06,A -85,B 0,C 180,E1 14445.322,E2 14445.322} C_VEL
LIN {X 0,Y 343.209,Z 834.236,A -85,B 0,C 180,E1 14443.666,E2 14443.666} C_VEL
LIN {X 0,Y 347.882,Z 815.095,A -85,B 0,C 180,E1 14442.316,E2 14442.316} C_VEL
LIN {X 0,Y 351.673,Z 795.599,A -85,B 0,C 180,E1 14441.235,E2 14441.235} C_VEL
LIN {X 0,Y 354.566,Z 775.461,A -85,B 0,C 180,E1 14440.39,E2 14440.39} C_VEL
LIN {X 0,Y 356.608,Z 753.633,A -85,B 0,C 180,E1 14439.734,E2 14439.734} C_VEL
LIN {X 0,Y 368.894,Z 536.076,A -85,B 0,C 180,E1 14435.558,E2 14435.558} C_VEL
LIN {X 0,Y 361.606,Z 523.659,A -85,B 0,C 180,E1 14433.006,E2 14433.006} C_VEL
LIN {X 0,Y 354.739,Z 512.766,A -85,B 0,C 180,E1 14430.3,E2 14430.3} C_VEL
LIN {X 0,Y 347.912,Z 502.382,A -85,B 0,C 180,E1 14427.191,E2 14427.191} C_VEL
LIN {X 0,Y 343.494,Z 496.172,A -85,B 0,C 180,E1 14424.874,E2 14424.874} C_VEL
LIN {X 0,Y 338.218,Z 488.823,A -85,B 0,C 180,E1 14421.596,E2 14421.596} C_VEL
LIN {X 0,Y 334.61,Z 483.857,A -85,B 0,C 180,E1 14418.828,E2 14418.828} C_VEL
LIN {X 0,Y 331.146,Z 479.157,A -85,B 0,C 180,E1 14415.409,E2 14415.409} C_VEL
LIN {X 0,Y 327.571,Z 474.054,A -85,B 0,C 180,E1 14409.133,E2 14409.133} C_VEL
LIN {X 0,Y 327.192,Z 473.669,A -85,B 0,C 180,E1 14403.68,E2 14403.68} C_VEL
LIN {X 0,Y 328.571,Z 474.67,A -85,B 0,C 180,E1 14399.826,E2 14399.826} C_VEL
LIN {X 0,Y 333.424,Z 480.721,A -85,B 0,C 180,E1 14393.63,E2 14393.63} C_VEL
LIN {X 0,Y 337.89,Z 486.327,A -85,B 0,C 180,E1 14390.032,E2 14390.032} C_VEL
LIN {X 0,Y 341.989,Z 491.618,A -85,B 0,C 180,E1 14387.377,E2 14387.377} C_VEL
LIN {X 0,Y 346.301,Z 497.372,A -85,B 0,C 180,E1 14384.982,E2 14384.982} C_VEL
LIN {X 0,Y 352.115,Z 505.367,A -85,B 0,C 180,E1 14382.184,E2 14382.184} C_VEL
LIN {X 0,Y 359.119,Z 515.586,A -85,B 0,C 180,E1 14379.251,E2 14379.251} C_VEL
LIN {X 0,Y 367.415,Z 528.694,A -85,B 0,C 180,E1 14376.207,E2 14376.207} C_VEL
LIN {X 0,Y 373.174,Z 538.512,A -85,B 0,C 180,E1 14374.297,E2 14374.297} C_VEL
LIN {X 0,Y 359.217,Z 740.845,A -85,B 0,C 180,E1 14370.003,E2 14370.003} C_VEL
LIN {X 0,Y 355.257,Z 796.184,A -85,B 0,C 180,E1 14368.768,E2 14368.768} C_VEL
LIN {X 0,Y 352.122,Z 819.667,A -85,B 0,C 180,E1 14368.05,E2 14368.05} C_VEL
LIN {X 0,Y 347.718,Z 843.315,A -85,B 0,C 180,E1 14367.103,E2 14367.103} C_VEL
LIN {X 0,Y 342.77,Z 865.362,A -85,B 0,C 180,E1 14365.938,E2 14365.938} C_VEL
LIN {X 0,Y 337.135,Z 886.641,A -85,B 0,C 180,E1 14364.499,E2 14364.499} C_VEL
LIN {X 0,Y 330.694,Z 908.372,A -85,B 0,C 180,E1 14362.673,E2 14362.673} C_VEL
LIN {X 0,Y 324.186,Z 928.638,A -85,B 0,C 180,E1 14360.588,E2 14360.588} C_VEL
LIN {X 0,Y 317.655,Z 947.372,A -85,B 0,C 180,E1 14358.244,E2 14358.244} C_VEL
LIN {X 0,Y 310.634,Z 966.732,A -85,B 0,C 180,E1 14355.345,E2 14355.345} C_VEL
LIN {X 0,Y 304.268,Z 984.162,A -85,B 0,C 180,E1 14352.223,E2 14352.223} C_VEL
LIN {X 0,Y 298.421,Z 1000.105,A -85,B 0,C 180,E1 14348.796,E2 14348.796} C_VEL
LIN {X 0,Y 292.911,Z 1015.911,A -85,B 0,C 180,E1 14344.755,E2 14344.755} C_VEL
LIN {X 0,Y 288.778,Z 1028.883,A -85,B 0,C 180,E1 14340.826,E2 14340.826} C_VEL
LIN {X 0,Y 285.534,Z 1040.389,A -85,B 0,C 180,E1 14336.63,E2 14336.63} C_VEL
LIN {X 0,Y 283.144,Z 1050.992,A -85,B 0,C 180,E1 14331.982,E2 14331.982} C_VEL
LIN {X 0,Y 281.942,Z 1058.456,A -85,B 0,C 180,E1 14327.971,E2 14327.971} C_VEL
LIN {X 0,Y 281.354,Z 1064.957,A -85,B 0,C 180,E1 14323.565,E2 14323.565} C_VEL
LIN {X 0,Y 281.27,Z 1069.095,A -85,B 0,C 180,E1 14319.825,E2 14319.825} C_VEL
LIN {X 0,Y 281.442,Z 1072.152,A -85,B 0,C 180,E1 14315.889,E2 14315.889} C_VEL
LIN {X 0,Y 281.59,Z 1073.599,A -85,B 0,C 180,E1 14312.035,E2 14312.035} C_VEL
LIN {X 0,Y 281.599,Z 1073.716,A -85,B 0,C 180,E1 14308.779,E2 14308.779} C_VEL
LIN {X 0,Y 281.495,Z 1072.71,A -85,B 0,C 180,E1 14305.314,E2 14305.314} C_VEL
LIN {X 0,Y 281.307,Z 1070.262,A -85,B 0,C 180,E1 14301.415,E2 14301.415} C_VEL
LIN {X 0,Y 281.32,Z 1065.973,A -85,B 0,C 180,E1 14297.27,E2 14297.27} C_VEL
LIN {X 0,Y 281.704,Z 1060.505,A -85,B 0,C 180,E1 14293.292,E2 14293.292} C_VEL
LIN {X 0,Y 282.818,Z 1052.663,A -85,B 0,C 180,E1 14288.862,E2 14288.862} C_VEL
LIN {X 0,Y 284.634,Z 1044.014,A -85,B 0,C 180,E1 14284.846,E2 14284.846} C_VEL
LIN {X 0,Y 287.507,Z 1033.054,A -85,B 0,C 180,E1 14280.636,E2 14280.636} C_VEL
LIN {X 0,Y 291.247,Z 1020.937,A -85,B 0,C 180,E1 14276.682,E2 14276.682} C_VEL
LIN {X 0,Y 296.059,Z 1006.678,A -85,B 0,C 180,E1 14272.805,E2 14272.805} C_VEL
LIN {X 0,Y 302.005,Z 990.121,A -85,B 0,C 180,E1 14269.011,E2 14269.011} C_VEL
LIN {X 0,Y 308.229,Z 973.343,A -85,B 0,C 180,E1 14265.778,E2 14265.778} C_VEL
LIN {X 0,Y 314.922,Z 954.883,A -85,B 0,C 180,E1 14262.826,E2 14262.826} C_VEL
LIN {X 0,Y 321.925,Z 934.98,A -85,B 0,C 180,E1 14260.177,E2 14260.177} C_VEL
LIN {X 0,Y 328.574,Z 915.128,A -85,B 0,C 180,E1 14257.987,E2 14257.987} C_VEL
LIN {X 0,Y 334.777,Z 894.722,A -85,B 0,C 180,E1 14256.148,E2 14256.148} C_VEL
LIN {X 0,Y 340.946,Z 872.193,A -85,B 0,C 180,E1 14254.506,E2 14254.506} C_VEL
LIN {X 0,Y 346.138,Z 850.592,A -85,B 0,C 180,E1 14253.253,E2 14253.253} C_VEL
LIN {X 0,Y 350.679,Z 827.668,A -85,B 0,C 180,E1 14252.248,E2 14252.248} C_VEL
LIN {X 0,Y 354.298,Z 803.536,A -85,B 0,C 180,E1 14251.451,E2 14251.451} C_VEL
LIN {X 0,Y 356.581,Z 778.954,A -85,B 0,C 180,E1 14250.835,E2 14250.835} C_VEL
LIN {X 0,Y 370.583,Z 574.243,A -85,B 0,C 180,E1 14246.454,E2 14246.454} C_VEL
LIN {X 0,Y 373.022,Z 538.281,A -85,B 0,C 180,E1 14245.693,E2 14245.693} C_VEL
LIN {X 0,Y 365.059,Z 524.976,A -85,B 0,C 180,E1 14243.015,E2 14243.015} C_VEL
LIN {X 0,Y 357.035,Z 512.575,A -85,B 0,C 180,E1 14239.977,E2 14239.977} C_VEL
LIN {X 0,Y 350.281,Z 502.914,A -85,B 0,C 180,E1 14237.055,E2 14237.055} C_VEL
LIN {X 0,Y 344.43,Z 494.89,A -85,B 0,C 180,E1 14234.113,E2 14234.113} C_VEL
LIN {X 0,Y 340.422,Z 489.639,A -85,B 0,C 180,E1 14231.778,E2 14231.778} C_VEL
LIN {X 0,Y 336.562,Z 484.752,A -85,B 0,C 180,E1 14229.145,E2 14229.145} C_VEL
LIN {X 0,Y 332.695,Z 479.849,A -85,B 0,C 180,E1 14225.864,E2 14225.864} C_VEL
LIN {X 0,Y 328.262,Z 474.337,A -85,B 0,C 180,E1 14219.999,E2 14219.999} C_VEL
LIN {X 0,Y 326.757,Z 473.438,A -85,B 0,C 180,E1 14214.556,E2 14214.556} C_VEL
LIN {X 0,Y 327.603,Z 474.17,A -85,B 0,C 180,E1 14209.981,E2 14209.981} C_VEL
LIN {X 0,Y 331.563,Z 479.808,A -85,B 0,C 180,E1 14203.802,E2 14203.802} C_VEL
LIN {X 0,Y 335.353,Z 484.908,A -85,B 0,C 180,E1 14200.311,E2 14200.311} C_VEL
LIN {X 0,Y 339.664,Z 490.917,A -85,B 0,C 180,E1 14197.226,E2 14197.226} C_VEL
LIN {X 0,Y 345.133,Z 498.383,A -85,B 0,C 180,E1 14194.058,E2 14194.058} C_VEL
LIN {X 0,Y 351.775,Z 508.314,A -85,B 0,C 180,E1 14190.826,E2 14190.826} C_VEL
LIN {X 0,Y 358.952,Z 519.39,A -85,B 0,C 180,E1 14187.857,E2 14187.857} C_VEL
LIN {X 0,Y 366.975,Z 532.768,A -85,B 0,C 180,E1 14184.955,E2 14184.955} C_VEL
LIN {X 0,Y 368.856,Z 536.423,A -85,B 0,C 180,E1 14184.313,E2 14184.313} C_VEL
LIN {X 0,Y 356.321,Z 756.684,A -85,B 0,C 180,E1 14180.091,E2 14180.091} C_VEL
LIN {X 0,Y 354.213,Z 777.483,A -85,B 0,C 180,E1 14179.436,E2 14179.436} C_VEL
LIN {X 0,Y 351.031,Z 798.546,A -85,B 0,C 180,E1 14178.514,E2 14178.514} C_VEL
LIN {X 0,Y 347.195,Z 817.852,A -85,B 0,C 180,E1 14177.409,E2 14177.409} C_VEL
LIN {X 0,Y 342.537,Z 836.452,A -85,B 0,C 180,E1 14176.056,E2 14176.056} C_VEL
LIN {X 0,Y 337.143,Z 854.608,A -85,B 0,C 180,E1 14174.42,E2 14174.42} C_VEL
LIN {X 0,Y 331.297,Z 871.716,A -85,B 0,C 180,E1 14172.535,E2 14172.535} C_VEL
LIN {X 0,Y 325.077,Z 887.819,A -85,B 0,C 180,E1 14170.374,E2 14170.374} C_VEL
LIN {X 0,Y 318.734,Z 902.597,A -85,B 0,C 180,E1 14167.941,E2 14167.941} C_VEL
LIN {X 0,Y 312.319,Z 916.405,A -85,B 0,C 180,E1 14165.188,E2 14165.188} C_VEL
LIN {X 0,Y 306.218,Z 928.865,A -85,B 0,C 180,E1 14162.156,E2 14162.156} C_VEL
LIN {X 0,Y 300.214,Z 940.454,A -85,B 0,C 180,E1 14158.659,E2 14158.659} C_VEL
LIN {X 0,Y 295.18,Z 949.975,A -85,B 0,C 180,E1 14155.05,E2 14155.05} C_VEL
LIN {X 0,Y 290.679,Z 958.508,A -85,B 0,C 180,E1 14150.961,E2 14150.961} C_VEL
LIN {X 0,Y 287.338,Z 965.166,A -85,B 0,C 180,E1 14146.787,E2 14146.787} C_VEL
LIN {X 0,Y 285.008,Z 970.16,A -85,B 0,C 180,E1 14142.563,E2 14142.563} C_VEL
LIN {X 0,Y 283.546,Z 973.634,A -85,B 0,C 180,E1 14138.109,E2 14138.109} C_VEL
LIN {X 0,Y 282.799,Z 975.573,A -85,B 0,C 180,E1 14133.649,E2 14133.649} C_VEL
LIN {X 0,Y 282.646,Z 976.061,A -85,B 0,C 180,E1 14129.189,E2 14129.189} C_VEL
LIN {X 0,Y 282.965,Z 975.215,A -85,B 0,C 180,E1 14124.932,E2 14124.932} C_VEL
LIN {X 0,Y 283.902,Z 972.752,A -85,B 0,C 180,E1 14120.444,E2 14120.444} C_VEL
LIN {X 0,Y 285.625,Z 968.753,A -85,B 0,C 180,E1 14116.022,E2 14116.022} C_VEL
LIN {X 0,Y 288.439,Z 962.999,A -85,B 0,C 180,E1 14111.612,E2 14111.612} C_VEL
LIN {X 0,Y 292.181,Z 955.733,A -85,B 0,C 180,E1 14107.463,E2 14107.463} C_VEL
LIN {X 0,Y 296.833,Z 946.986,A -85,B 0,C 180,E1 14103.6,E2 14103.6} C_VEL
LIN {X 0,Y 302.198,Z 936.715,A -85,B 0,C 180,E1 14100.026,E2 14100.026} C_VEL
LIN {X 0,Y 308.154,Z 925.039,A -85,B 0,C 180,E1 14096.746,E2 14096.746} C_VEL
LIN {X 0,Y 314.515,Z 911.952,A -85,B 0,C 180,E1 14093.75,E2 14093.75} C_VEL
LIN {X 0,Y 319.035,Z 902.075,A -85,B 0,C 180,E1 14091.858,E2 14091.858} C_VEL
LIN {X 0,Y 320.611,Z 897.039,A -85,B 0,C 180,E1 14090.832,E2 14090.832} C_VEL
LIN {X 0,Y 321.928,Z 884.542,A -85,B 0,C 180,E1 14088.031,E2 14088.031} C_VEL
LIN {X 0,Y 323.506,Z 878.903,A -85,B 0,C 180,E1 14087.132,E2 14087.132} C_VEL
LIN {X 0,Y 329.927,Z 861.7,A -85,B 0,C 180,E1 14085.08,E2 14085.08} C_VEL
LIN {X 0,Y 335.608,Z 844.028,A -85,B 0,C 180,E1 14083.369,E2 14083.369} C_VEL
LIN {X 0,Y 340.934,Z 824.583,A -85,B 0,C 180,E1 14081.848,E2 14081.848} C_VEL
LIN {X 0,Y 345.264,Z 805.306,A -85,B 0,C 180,E1 14080.647,E2 14080.647} C_VEL
LIN {X 0,Y 348.749,Z 784.994,A -85,B 0,C 180,E1 14079.673,E2 14079.673} C_VEL
LIN {X 0,Y 351.223,Z 764.196,A -85,B 0,C 180,E1 14078.94,E2 14078.94} C_VEL
LIN {X 0,Y 353.023,Z 737.894,A -85,B 0,C 180,E1 14078.329,E2 14078.329} C_VEL
LIN {X 0,Y 364.746,Z 540.389,A -85,B 0,C 180,E1 14074.572,E2 14074.572} C_VEL
LIN {X 0,Y 357.55,Z 527.944,A -85,B 0,C 180,E1 14071.906,E2 14071.906} C_VEL
LIN {X 0,Y 350.545,Z 516.763,A -85,B 0,C 180,E1 14068.959,E2 14068.959} C_VEL
LIN {X 0,Y 344.627,Z 507.837,A -85,B 0,C 180,E1 14066.075,E2 14066.075} C_VEL
LIN {X 0,Y 340.342,Z 501.476,A -85,B 0,C 180,E1 14063.642,E2 14063.642} C_VEL
LIN {X 0,Y 336.342,Z 496.009,A -85,B 0,C 180,E1 14061,E2 14061} C_VEL
LIN {X 0,Y 333.172,Z 491.47,A -85,B 0,C 180,E1 14058.458,E2 14058.458} C_VEL
LIN {X 0,Y 329.898,Z 486.924,A -85,B 0,C 180,E1 14055.109,E2 14055.109} C_VEL
LIN {X 0,Y 326.56,Z 481.959,A -85,B 0,C 180,E1 14048.984,E2 14048.984} C_VEL
LIN {X 0,Y 326.212,Z 481.609,A -85,B 0,C 180,E1 14043.691,E2 14043.691} C_VEL
LIN {X 0,Y 327.58,Z 482.658,A -85,B 0,C 180,E1 14039.826,E2 14039.826} C_VEL
LIN {X 0,Y 332.059,Z 488.382,A -85,B 0,C 180,E1 14033.951,E2 14033.951} C_VEL
LIN {X 0,Y 336.407,Z 494.012,A -85,B 0,C 180,E1 14030.333,E2 14030.333} C_VEL
LIN {X 0,Y 340.353,Z 499.237,A -85,B 0,C 180,E1 14027.703,E2 14027.703} C_VEL
LIN {X 0,Y 344.58,Z 505.016,A -85,B 0,C 180,E1 14025.292,E2 14025.292} C_VEL
LIN {X 0,Y 350.113,Z 512.847,A -85,B 0,C 180,E1 14022.551,E2 14022.551} C_VEL
LIN {X 0,Y 356.812,Z 522.825,A -85,B 0,C 180,E1 14019.668,E2 14019.668} C_VEL
LIN {X 0,Y 364.856,Z 535.89,A -85,B 0,C 180,E1 14016.63,E2 14016.63} C_VEL
LIN {X 0,Y 368.766,Z 542.826,A -85,B 0,C 180,E1 14015.273,E2 14015.273} C_VEL
LIN {X 0,Y 354.289,Z 746.122,A -85,B 0,C 180,E1 14010.948,E2 14010.948} C_VEL
LIN {X 0,Y 350.603,Z 795.634,A -85,B 0,C 180,E1 14009.836,E2 14009.836} C_VEL
LIN {X 0,Y 347.394,Z 819.046,A -85,B 0,C 180,E1 14009.12,E2 14009.12} C_VEL
LIN {X 0,Y 342.96,Z 842.241,A -85,B 0,C 180,E1 14008.194,E2 14008.194} C_VEL
LIN {X 0,Y 338.173,Z 863.108,A -85,B 0,C 180,E1 14007.108,E2 14007.108} C_VEL
LIN {X 0,Y 332.25,Z 884.847,A -85,B 0,C 180,E1 14005.655,E2 14005.655} C_VEL
LIN {X 0,Y 325.355,Z 907.318,A -85,B 0,C 180,E1 14003.775,E2 14003.775} C_VEL
LIN {X 0,Y 318.587,Z 927.562,A -85,B 0,C 180,E1 14001.685,E2 14001.685} C_VEL
LIN {X 0,Y 311.542,Z 946.94,A -85,B 0,C 180,E1 13999.237,E2 13999.237} C_VEL
LIN {X 0,Y 304.237,Z 966.169,A -85,B 0,C 180,E1 13996.305,E2 13996.305} C_VEL
LIN {X 0,Y 297.708,Z 983.121,A -85,B 0,C 180,E1 13993.215,E2 13993.215} C_VEL
LIN {X 0,Y 291.443,Z 999.363,A -85,B 0,C 180,E1 13989.652,E2 13989.652} C_VEL
LIN {X 0,Y 285.899,Z 1014.344,A -85,B 0,C 180,E1 13985.736,E2 13985.736} C_VEL
LIN {X 0,Y 281.473,Z 1027.341,A -85,B 0,C 180,E1 13981.718,E2 13981.718} C_VEL
LIN {X 0,Y 277.903,Z 1039.168,A -85,B 0,C 180,E1 13977.295,E2 13977.295} C_VEL
LIN {X 0,Y 275.306,Z 1049.938,A -85,B 0,C 180,E1 13972.417,E2 13972.417} C_VEL
LIN {X 0,Y 273.983,Z 1057.731,A -85,B 0,C 180,E1 13968.071,E2 13968.071} C_VEL
LIN {X 0,Y 273.407,Z 1064.049,A -85,B 0,C 180,E1 13963.536,E2 13963.536} C_VEL
LIN {X 0,Y 273.348,Z 1068.092,A -85,B 0,C 180,E1 13959.687,E2 13959.687} C_VEL
LIN {X 0,Y 273.548,Z 1070.98,A -85,B 0,C 180,E1 13955.664,E2 13955.664} C_VEL
LIN {X 0,Y 273.712,Z 1072.264,A -85,B 0,C 180,E1 13951.884,E2 13951.884} C_VEL
LIN {X 0,Y 273.718,Z 1072.322,A -85,B 0,C 180,E1 13948.535,E2 13948.535} C_VEL
LIN {X 0,Y 273.578,Z 1071.246,A -85,B 0,C 180,E1 13944.968,E2 13944.968} C_VEL
LIN {X 0,Y 273.362,Z 1068.674,A -85,B 0,C 180,E1 13940.949,E2 13940.949} C_VEL
LIN {X 0,Y 273.393,Z 1064.553,A -85,B 0,C 180,E1 13936.894,E2 13936.894} C_VEL
LIN {X 0,Y 273.847,Z 1058.747,A -85,B 0,C 180,E1 13932.579,E2 13932.579} C_VEL
LIN {X 0,Y 275.131,Z 1050.765,A -85,B 0,C 180,E1 13928.018,E2 13928.018} C_VEL
LIN {X 0,Y 277.28,Z 1041.537,A -85,B 0,C 180,E1 13923.67,E2 13923.67} C_VEL
LIN {X 0,Y 280.487,Z 1030.323,A -85,B 0,C 180,E1 13919.352,E2 13919.352} C_VEL
LIN {X 0,Y 285.121,Z 1016.479,A -85,B 0,C 180,E1 13914.892,E2 13914.892} C_VEL
LIN {X 0,Y 290.483,Z 1001.9,A -85,B 0,C 180,E1 13910.957,E2 13910.957} C_VEL
LIN {X 0,Y 296.629,Z 985.771,A -85,B 0,C 180,E1 13907.349,E2 13907.349} C_VEL
LIN {X 0,Y 303.578,Z 967.752,A -85,B 0,C 180,E1 13903.974,E2 13903.974} C_VEL
LIN {X 0,Y 310.59,Z 949.469,A -85,B 0,C 180,E1 13901.123,E2 13901.123} C_VEL
LIN {X 0,Y 317.276,Z 931.022,A -85,B 0,C 180,E1 13898.742,E2 13898.742} C_VEL
LIN {X 0,Y 324.506,Z 909.738,A -85,B 0,C 180,E1 13896.468,E2 13896.468} C_VEL
LIN {X 0,Y 330.834,Z 889.6,A -85,B 0,C 180,E1 13894.709,E2 13894.709} C_VEL
LIN {X 0,Y 336.58,Z 868.781,A -85,B 0,C 180,E1 13893.254,E2 13893.254} C_VEL
LIN {X 0,Y 342.286,Z 844.946,A -85,B 0,C 180,E1 13891.941,E2 13891.941} C_VEL
LIN {X 0,Y 346.81,Z 822.215,A -85,B 0,C 180,E1 13890.997,E2 13890.997} C_VEL
LIN {X 0,Y 350.12,Z 798.845,A -85,B 0,C 180,E1 13890.266,E2 13890.266} C_VEL
LIN {X 0,Y 352.784,Z 766.633,A -85,B 0,C 180,E1 13889.508,E2 13889.508} C_VEL
LIN {X 0,Y 367.519,Z 558.555,A -85,B 0,C 180,E1 13885.063,E2 13885.063} C_VEL
LIN {X 0,Y 368.564,Z 542.315,A -85,B 0,C 180,E1 13884.694,E2 13884.694} C_VEL
LIN {X 0,Y 361.15,Z 529.939,A -85,B 0,C 180,E1 13882.075,E2 13882.075} C_VEL
LIN {X 0,Y 354.404,Z 519.27,A -85,B 0,C 180,E1 13879.402,E2 13879.402} C_VEL
LIN {X 0,Y 347.516,Z 509.201,A -85,B 0,C 180,E1 13876.291,E2 13876.291} C_VEL
LIN {X 0,Y 342.381,Z 502.054,A -85,B 0,C 180,E1 13873.596,E2 13873.596} C_VEL
LIN {X 0,Y 338.623,Z 497.018,A -85,B 0,C 180,E1 13871.323,E2 13871.323} C_VEL
LIN {X 0,Y 335.105,Z 492.417,A -85,B 0,C 180,E1 13868.839,E2 13868.839} C_VEL
LIN {X 0,Y 331.336,Z 487.568,A -85,B 0,C 180,E1 13865.541,E2 13865.541} C_VEL
LIN {X 0,Y 327.187,Z 482.212,A -85,B 0,C 180,E1 13859.824,E2 13859.824} C_VEL
LIN {X 0,Y 325.787,Z 481.373,A -85,B 0,C 180,E1 13854.187,E2 13854.187} C_VEL
LIN {X 0,Y 326.633,Z 482.189,A -85,B 0,C 180,E1 13849.951,E2 13849.951} C_VEL
LIN {X 0,Y 330.299,Z 487.525,A -85,B 0,C 180,E1 13844.1,E2 13844.1} C_VEL
LIN {X 0,Y 333.992,Z 492.668,A -85,B 0,C 180,E1 13840.591,E2 13840.591} C_VEL
LIN {X 0,Y 338.089,Z 498.505,A -85,B 0,C 180,E1 13837.573,E2 13837.573} C_VEL
LIN {X 0,Y 343.37,Z 505.93,A -85,B 0,C 180,E1 13834.425,E2 13834.425} C_VEL
LIN {X 0,Y 349.554,Z 515.366,A -85,B 0,C 180,E1 13831.325,E2 13831.325} C_VEL
LIN {X 0,Y 356.578,Z 526.475,A -85,B 0,C 180,E1 13828.328,E2 13828.328} C_VEL
LIN {X 0,Y 364.14,Z 539.4,A -85,B 0,C 180,E1 13825.505,E2 13825.505} C_VEL
LIN {X 0,Y 364.618,Z 540.676,A -85,B 0,C 180,E1 13825.322,E2 13825.322} C_VEL
LIN {X 0,Y 351.749,Z 757.342,A -85,B 0,C 180,E1 13821.148,E2 13821.148} C_VEL
LIN {X 0,Y 349.557,Z 778.219,A -85,B 0,C 180,E1 13820.489,E2 13820.489} C_VEL
LIN {X 0,Y 346.216,Z 799.559,A -85,B 0,C 180,E1 13819.551,E2 13819.551} C_VEL
LIN {X 0,Y 342.176,Z 819.133,A -85,B 0,C 180,E1 13818.422,E2 13818.422} C_VEL
LIN {X 0,Y 337.354,Z 837.748,A -85,B 0,C 180,E1 13817.06,E2 13817.06} C_VEL
LIN {X 0,Y 331.841,Z 855.66,A -85,B 0,C 180,E1 13815.434,E2 13815.434} C_VEL
LIN {X 0,Y 325.817,Z 872.706,A -85,B 0,C 180,E1 13813.547,E2 13813.547} C_VEL
LIN {X 0,Y 319.324,Z 888.944,A -85,B 0,C 180,E1 13811.352,E2 13811.352} C_VEL
LIN {X 0,Y 313,Z 903.158,A -85,B 0,C 180,E1 13808.999,E2 13808.999} C_VEL
LIN {X 0,Y 305.91,Z 917.87,A -85,B 0,C 180,E1 13806.039,E2 13806.039} C_VEL
LIN {X 0,Y 299.557,Z 930.294,A -85,B 0,C 180,E1 13802.961,E2 13802.961} C_VEL
LIN {X 0,Y 293.296,Z 941.876,A -85,B 0,C 180,E1 13799.4,E2 13799.4} C_VEL
LIN {X 0,Y 288.023,Z 951.375,A -85,B 0,C 180,E1 13795.718,E2 13795.718} C_VEL
LIN {X 0,Y 283.29,Z 959.897,A -85,B 0,C 180,E1 13791.535,E2 13791.535} C_VEL
LIN {X 0,Y 279.761,Z 966.547,A -85,B 0,C 180,E1 13787.256,E2 13787.256} C_VEL
LIN {X 0,Y 277.286,Z 971.537,A -85,B 0,C 180,E1 13782.919,E2 13782.919} C_VEL
LIN {X 0,Y 275.725,Z 975.006,A -85,B 0,C 180,E1 13778.34,E2 13778.34} C_VEL
LIN {X 0,Y 274.949,Z 976.883,A -85,B 0,C 180,E1 13773.962,E2 13773.962} C_VEL
LIN {X 0,Y 274.759,Z 977.467,A -85,B 0,C 180,E1 13769.583,E2 13769.583} C_VEL
LIN {X 0,Y 275.044,Z 976.692,A -85,B 0,C 180,E1 13765.204,E2 13765.204} C_VEL
LIN {X 0,Y 275.916,Z 974.542,A -85,B 0,C 180,E1 13760.825,E2 13760.825} C_VEL
LIN {X 0,Y 277.631,Z 970.784,A -85,B 0,C 180,E1 13756.25,E2 13756.25} C_VEL
LIN {X 0,Y 280.314,Z 965.619,A -85,B 0,C 180,E1 13751.921,E2 13751.921} C_VEL
LIN {X 0,Y 284.239,Z 958.298,A -85,B 0,C 180,E1 13747.454,E2 13747.454} C_VEL
LIN {X 0,Y 288.954,Z 949.77,A -85,B 0,C 180,E1 13743.489,E2 13743.489} C_VEL
LIN {X 0,Y 294.413,Z 939.865,A -85,B 0,C 180,E1 13739.826,E2 13739.826} C_VEL
LIN {X 0,Y 300.498,Z 928.609,A -85,B 0,C 180,E1 13736.472,E2 13736.472} C_VEL
LIN {X 0,Y 306.984,Z 915.921,A -85,B 0,C 180,E1 13733.413,E2 13733.413} C_VEL
LIN {X 0,Y 313.73,Z 901.745,A -85,B 0,C 180,E1 13730.638,E2 13730.638} C_VEL
LIN {X 0,Y 320.576,Z 886.077,A -85,B 0,C 180,E1 13728.129,E2 13728.129} C_VEL
LIN {X 0,Y 323.506,Z 878.903,A -85,B 0,C 180,E1 13727.132,E2 13727.132} C_VEL
LIN {X 0,Y 325.069,Z 873.237,A -85,B 0,C 180,E1 13726.264,E2 13726.264} C_VEL
LIN {X 0,Y 326.64,Z 858.903,A -85,B 0,C 180,E1 13723.786,E2 13723.786} C_VEL
LIN {X 0,Y 328.14,Z 852.675,A -85,B 0,C 180,E1 13723.009,E2 13723.009} C_VEL
LIN {X 0,Y 333.749,Z 834.167,A -85,B 0,C 180,E1 13721.416,E2 13721.416} C_VEL
LIN {X 0,Y 338.807,Z 814.171,A -85,B 0,C 180,E1 13720.042,E2 13720.042} C_VEL
LIN {X 0,Y 342.798,Z 794.371,A -85,B 0,C 180,E1 13718.976,E2 13718.976} C_VEL
LIN {X 0,Y 345.742,Z 774.39,A -85,B 0,C 180,E1 13718.164,E2 13718.164} C_VEL
LIN {X 0,Y 347.718,Z 753.454,A -85,B 0,C 180,E1 13717.556,E2 13717.556} C_VEL
LIN {X 0,Y 360.617,Z 544.657,A -85,B 0,C 180,E1 13713.536,E2 13713.536} C_VEL
LIN {X 0,Y 353.79,Z 532.691,A -85,B 0,C 180,E1 13710.861,E2 13710.861} C_VEL
LIN {X 0,Y 346.524,Z 520.899,A -85,B 0,C 180,E1 13707.588,E2 13707.588} C_VEL
LIN {X 0,Y 340.633,Z 511.919,A -85,B 0,C 180,E1 13704.449,E2 13704.449} C_VEL
LIN {X 0,Y 335.28,Z 504.116,A -85,B 0,C 180,E1 13700.969,E2 13700.969} C_VEL
LIN {X 0,Y 331.84,Z 499.185,A -85,B 0,C 180,E1 13698.171,E2 13698.171} C_VEL
LIN {X 0,Y 328.66,Z 494.688,A -85,B 0,C 180,E1 13694.807,E2 13694.807} C_VEL
LIN {X 0,Y 325.595,Z 489.918,A -85,B 0,C 180,E1 13689.011,E2 13689.011} C_VEL
LIN {X 0,Y 325.239,Z 489.55,A -85,B 0,C 180,E1 13683.702,E2 13683.702} C_VEL
LIN {X 0,Y 326.505,Z 490.524,A -85,B 0,C 180,E1 13680.001,E2 13680.001} C_VEL
LIN {X 0,Y 330.794,Z 496.192,A -85,B 0,C 180,E1 13674.189,E2 13674.189} C_VEL
LIN {X 0,Y 334.934,Z 501.695,A -85,B 0,C 180,E1 13670.637,E2 13670.637} C_VEL
LIN {X 0,Y 338.665,Z 506.753,A -85,B 0,C 180,E1 13668.074,E2 13668.074} C_VEL
LIN {X 0,Y 342.715,Z 512.439,A -85,B 0,C 180,E1 13665.685,E2 13665.685} C_VEL
LIN {X 0,Y 348.048,Z 520.193,A -85,B 0,C 180,E1 13662.962,E2 13662.962} C_VEL
LIN {X 0,Y 354.529,Z 530.065,A -85,B 0,C 180,E1 13660.091,E2 13660.091} C_VEL
LIN {X 0,Y 362.12,Z 542.73,A -85,B 0,C 180,E1 13657.131,E2 13657.131} C_VEL
LIN {X 0,Y 364.468,Z 547.08,A -85,B 0,C 180,E1 13656.274,E2 13656.274} C_VEL
LIN {X 0,Y 349.365,Z 752.914,A -85,B 0,C 180,E1 13651.887,E2 13651.887} C_VEL
LIN {X 0,Y 346.038,Z 795.391,A -85,B 0,C 180,E1 13650.924,E2 13650.924} C_VEL
LIN {X 0,Y 342.773,Z 818.539,A -85,B 0,C 180,E1 13650.215,E2 13650.215} C_VEL
LIN {X 0,Y 338.16,Z 841.934,A -85,B 0,C 180,E1 13649.281,E2 13649.281} C_VEL
LIN {X 0,Y 333.069,Z 863.288,A -85,B 0,C 180,E1 13648.164,E2 13648.164} C_VEL
LIN {X 0,Y 326.993,Z 884.799,A -85,B 0,C 180,E1 13646.716,E2 13646.716} C_VEL
LIN {X 0,Y 320.147,Z 906.277,A -85,B 0,C 180,E1 13644.912,E2 13644.912} C_VEL
LIN {X 0,Y 313.114,Z 926.499,A -85,B 0,C 180,E1 13642.819,E2 13642.819} C_VEL
LIN {X 0,Y 305.895,Z 945.53,A -85,B 0,C 180,E1 13640.404,E2 13640.404} C_VEL
LIN {X 0,Y 298.387,Z 964.503,A -85,B 0,C 180,E1 13637.493,E2 13637.493} C_VEL
LIN {X 0,Y 291.348,Z 981.862,A -85,B 0,C 180,E1 13634.298,E2 13634.298} C_VEL
LIN {X 0,Y 284.725,Z 998.133,A -85,B 0,C 180,E1 13630.667,E2 13630.667} C_VEL
LIN {X 0,Y 278.689,Z 1013.504,A -85,B 0,C 180,E1 13626.553,E2 13626.553} C_VEL
LIN {X 0,Y 273.801,Z 1027.022,A -85,B 0,C 180,E1 13622.219,E2 13622.219} C_VEL
LIN {X 0,Y 270.164,Z 1038.439,A -85,B 0,C 180,E1 13617.796,E2 13617.796} C_VEL
LIN {X 0,Y 267.573,Z 1048.46,A -85,B 0,C 180,E1 13613.102,E2 13613.102} C_VEL
LIN {X 0,Y 266.13,Z 1056.278,A -85,B 0,C 180,E1 13608.624,E2 13608.624} C_VEL
LIN {X 0,Y 265.478,Z 1062.626,A -85,B 0,C 180,E1 13603.948,E2 13603.948} C_VEL
LIN {X 0,Y 265.424,Z 1066.495,A -85,B 0,C 180,E1 13600.198,E2 13600.198} C_VEL
LIN {X 0,Y 265.622,Z 1069.504,A -85,B 0,C 180,E1 13596.05,E2 13596.05} C_VEL
LIN {X 0,Y 265.811,Z 1070.865,A -85,B 0,C 180,E1 13592.156,E2 13592.156} C_VEL
LIN {X 0,Y 265.833,Z 1070.984,A -85,B 0,C 180,E1 13588.707,E2 13588.707} C_VEL
LIN {X 0,Y 265.703,Z 1070.049,A -85,B 0,C 180,E1 13585.251,E2 13585.251} C_VEL
LIN {X 0,Y 265.473,Z 1067.778,A -85,B 0,C 180,E1 13581.335,E2 13581.335} C_VEL
LIN {X 0,Y 265.447,Z 1063.643,A -85,B 0,C 180,E1 13576.938,E2 13576.938} C_VEL
LIN {X 0,Y 265.855,Z 1058.242,A -85,B 0,C 180,E1 13572.716,E2 13572.716} C_VEL
LIN {X 0,Y 267.205,Z 1050.132,A -85,B 0,C 180,E1 13567.794,E2 13567.794} C_VEL
LIN {X 0,Y 269.432,Z 1041.016,A -85,B 0,C 180,E1 13563.318,E2 13563.318} C_VEL
LIN {X 0,Y 272.774,Z 1029.987,A -85,B 0,C 180,E1 13558.879,E2 13558.879} C_VEL
LIN {X 0,Y 277.345,Z 1017.085,A -85,B 0,C 180,E1 13554.519,E2 13554.519} C_VEL
LIN {X 0,Y 282.542,Z 1003.501,A -85,B 0,C 180,E1 13550.695,E2 13550.695} C_VEL
LIN {X 0,Y 289.201,Z 986.969,A -85,B 0,C 180,E1 13546.799,E2 13546.799} C_VEL
LIN {X 0,Y 296.136,Z 969.967,A -85,B 0,C 180,E1 13543.454,E2 13543.454} C_VEL
LIN {X 0,Y 303.312,Z 952.065,A -85,B 0,C 180,E1 13540.55,E2 13540.55} C_VEL
LIN {X 0,Y 310.839,Z 932.399,A -85,B 0,C 180,E1 13537.906,E2 13537.906} C_VEL
LIN {X 0,Y 317.842,Z 912.994,A -85,B 0,C 180,E1 13535.746,E2 13535.746} C_VEL
LIN {X 0,Y 324.592,Z 892.365,A -85,B 0,C 180,E1 13533.885,E2 13533.885} C_VEL
LIN {X 0,Y 331.112,Z 870.075,A -85,B 0,C 180,E1 13532.272,E2 13532.272} C_VEL
LIN {X 0,Y 336.761,Z 847.828,A -85,B 0,C 180,E1 13531.003,E2 13531.003} C_VEL
LIN {X 0,Y 341.524,Z 825.059,A -85,B 0,C 180,E1 13530.028,E2 13530.028} C_VEL
LIN {X 0,Y 345.164,Z 801.596,A -85,B 0,C 180,E1 13529.263,E2 13529.263} C_VEL
LIN {X 0,Y 347.591,Z 776.481,A -85,B 0,C 180,E1 13528.638,E2 13528.638} C_VEL
LIN {X 0,Y 362.672,Z 569.782,A -85,B 0,C 180,E1 13524.208,E2 13524.208} C_VEL
LIN {X 0,Y 364.311,Z 546.666,A -85,B 0,C 180,E1 13523.707,E2 13523.707} C_VEL
LIN {X 0,Y 357.17,Z 534.47,A -85,B 0,C 180,E1 13521.04,E2 13521.04} C_VEL
LIN {X 0,Y 350.006,Z 523.127,A -85,B 0,C 180,E1 13518.013,E2 13518.013} C_VEL
LIN {X 0,Y 343.446,Z 513.553,A -85,B 0,C 180,E1 13514.8,E2 13514.8} C_VEL
LIN {X 0,Y 340.083,Z 508.856,A -85,B 0,C 180,E1 13512.911,E2 13512.911} C_VEL
LIN {X 0,Y 336.974,Z 504.535,A -85,B 0,C 180,E1 13510.946,E2 13510.946} C_VEL
LIN {X 0,Y 333.548,Z 499.965,A -85,B 0,C 180,E1 13508.446,E2 13508.446} C_VEL
LIN {X 0,Y 329.995,Z 495.289,A -85,B 0,C 180,E1 13505.215,E2 13505.215} C_VEL
LIN {X 0,Y 326.114,Z 490.095,A -85,B 0,C 180,E1 13499.648,E2 13499.648} C_VEL
LIN {X 0,Y 324.823,Z 489.313,A -85,B 0,C 180,E1 13493.992,E2 13493.992} C_VEL
LIN {X 0,Y 325.604,Z 490.081,A -85,B 0,C 180,E1 13490.097,E2 13490.097} C_VEL
LIN {X 0,Y 329.114,Z 495.387,A -85,B 0,C 180,E1 13484.312,E2 13484.312} C_VEL
LIN {X 0,Y 332.541,Z 500.244,A -85,B 0,C 180,E1 13480.959,E2 13480.959} C_VEL
LIN {X 0,Y 336.528,Z 506.092,A -85,B 0,C 180,E1 13477.923,E2 13477.923} C_VEL
LIN {X 0,Y 341.553,Z 513.35,A -85,B 0,C 180,E1 13474.836,E2 13474.836} C_VEL
LIN {X 0,Y 347.448,Z 522.551,A -85,B 0,C 180,E1 13471.792,E2 13471.792} C_VEL
LIN {X 0,Y 354.234,Z 533.557,A -85,B 0,C 180,E1 13468.805,E2 13468.805} C_VEL
LIN {X 0,Y 360.521,Z 544.602,A -85,B 0,C 180,E1 13466.361,E2 13466.361} C_VEL
LIN {X 0,Y 347.291,Z 758.103,A -85,B 0,C 180,E1 13462.23,E2 13462.23} C_VEL
LIN {X 0,Y 345.021,Z 778.94,A -85,B 0,C 180,E1 13461.57,E2 13461.57} C_VEL
LIN {X 0,Y 341.517,Z 800.567,A -85,B 0,C 180,E1 13460.617,E2 13460.617} C_VEL
LIN {X 0,Y 337.344,Z 820.1,A -85,B 0,C 180,E1 13459.486,E2 13459.486} C_VEL
LIN {X 0,Y 332.2,Z 839.313,A -85,B 0,C 180,E1 13458.073,E2 13458.073} C_VEL
LIN {X 0,Y 326.557,Z 856.966,A -85,B 0,C 180,E1 13456.456,E2 13456.456} C_VEL
LIN {X 0,Y 320.185,Z 874.33,A -85,B 0,C 180,E1 13454.512,E2 13454.512} C_VEL
LIN {X 0,Y 313.479,Z 890.523,A -85,B 0,C 180,E1 13452.299,E2 13452.299} C_VEL
LIN {X 0,Y 306.48,Z 905.617,A -85,B 0,C 180,E1 13449.75,E2 13449.75} C_VEL
LIN {X 0,Y 299.57,Z 919.327,A -85,B 0,C 180,E1 13446.926,E2 13446.926} C_VEL
LIN {X 0,Y 292.958,Z 931.721,A -85,B 0,C 180,E1 13443.802,E2 13443.802} C_VEL
LIN {X 0,Y 286.431,Z 943.297,A -85,B 0,C 180,E1 13440.177,E2 13440.177} C_VEL
LIN {X 0,Y 280.906,Z 952.778,A -85,B 0,C 180,E1 13436.419,E2 13436.419} C_VEL
LIN {X 0,Y 275.93,Z 961.285,A -85,B 0,C 180,E1 13432.139,E2 13432.139} C_VEL
LIN {X 0,Y 272.203,Z 967.925,A -85,B 0,C 180,E1 13427.751,E2 13427.751} C_VEL
LIN {X 0,Y 269.575,Z 972.912,A -85,B 0,C 180,E1 13423.295,E2 13423.295} C_VEL
LIN {X 0,Y 267.908,Z 976.376,A -85,B 0,C 180,E1 13418.586,E2 13418.586} C_VEL
LIN {X 0,Y 267.082,Z 978.249,A -85,B 0,C 180,E1 13414.079,E2 13414.079} C_VEL
LIN {X 0,Y 266.877,Z 978.832,A -85,B 0,C 180,E1 13409.571,E2 13409.571} C_VEL
LIN {X 0,Y 267.181,Z 978.058,A -85,B 0,C 180,E1 13405.062,E2 13405.062} C_VEL
LIN {X 0,Y 268.113,Z 975.913,A -85,B 0,C 180,E1 13400.556,E2 13400.556} C_VEL
LIN {X 0,Y 269.944,Z 972.16,A -85,B 0,C 180,E1 13395.85,E2 13395.85} C_VEL
LIN {X 0,Y 272.789,Z 967.001,A -85,B 0,C 180,E1 13391.404,E2 13391.404} C_VEL
LIN {X 0,Y 276.932,Z 959.682,A -85,B 0,C 180,E1 13386.825,E2 13386.825} C_VEL
LIN {X 0,Y 281.884,Z 951.166,A -85,B 0,C 180,E1 13382.769,E2 13382.769} C_VEL
LIN {X 0,Y 287.93,Z 940.699,A -85,B 0,C 180,E1 13378.841,E2 13378.841} C_VEL
LIN {X 0,Y 294.318,Z 929.34,A -85,B 0,C 180,E1 13375.435,E2 13375.435} C_VEL
LIN {X 0,Y 301.113,Z 916.587,A -85,B 0,C 180,E1 13372.339,E2 13372.339} C_VEL
LIN {X 0,Y 308.149,Z 902.294,A -85,B 0,C 180,E1 13369.538,E2 13369.538} C_VEL
LIN {X 0,Y 315.264,Z 886.498,A -85,B 0,C 180,E1 13367.01,E2 13367.01} C_VEL
LIN {X 0,Y 321.825,Z 870.375,A -85,B 0,C 180,E1 13364.898,E2 13364.898} C_VEL
LIN {X 0,Y 328.14,Z 852.675,A -85,B 0,C 180,E1 13363.009,E2 13363.009} C_VEL
LIN {X 0,Y 329.659,Z 846.354,A -85,B 0,C 180,E1 13362.268,E2 13362.268} C_VEL
LIN {X 0,Y 330.862,Z 830.534,A -85,B 0,C 180,E1 13360.123,E2 13360.123} C_VEL
LIN {X 0,Y 332.027,Z 823.787,A -85,B 0,C 180,E1 13359.501,E2 13359.501} C_VEL
LIN {X 0,Y 336.639,Z 803.653,A -85,B 0,C 180,E1 13358.292,E2 13358.292} C_VEL
LIN {X 0,Y 340.24,Z 783.266,A -85,B 0,C 180,E1 13357.352,E2 13357.352} C_VEL
LIN {X 0,Y 342.775,Z 762.168,A -85,B 0,C 180,E1 13356.645,E2 13356.645} C_VEL
LIN {X 0,Y 344.873,Z 730.956,A -85,B 0,C 180,E1 13355.969,E2 13355.969} C_VEL
LIN {X 0,Y 356.606,Z 548.961,A -85,B 0,C 180,E1 13352.475,E2 13352.475} C_VEL
LIN {X 0,Y 350.232,Z 537.639,A -85,B 0,C 180,E1 13349.832,E2 13349.832} C_VEL
LIN {X 0,Y 343.91,Z 527.238,A -85,B 0,C 180,E1 13346.832,E2 13346.832} C_VEL
LIN {X 0,Y 338.452,Z 518.741,A -85,B 0,C 180,E1 13343.782,E2 13343.782} C_VEL
LIN {X 0,Y 333.538,Z 511.423,A -85,B 0,C 180,E1 13340.441,E2 13340.441} C_VEL
LIN {X 0,Y 330.423,Z 506.798,A -85,B 0,C 180,E1 13337.796,E2 13337.796} C_VEL
LIN {X 0,Y 327.431,Z 502.449,A -85,B 0,C 180,E1 13334.502,E2 13334.502} C_VEL
LIN {X 0,Y 324.577,Z 497.822,A -85,B 0,C 180,E1 13328.861,E2 13328.861} C_VEL
LIN {X 0,Y 324.298,Z 497.516,A -85,B 0,C 180,E1 13323.536,E2 13323.536} C_VEL
LIN {X 0,Y 325.436,Z 498.39,A -85,B 0,C 180,E1 13320.177,E2 13320.177} C_VEL
LIN {X 0,Y 329.536,Z 503.998,A -85,B 0,C 180,E1 13314.429,E2 13314.429} C_VEL
LIN {X 0,Y 333.468,Z 509.375,A -85,B 0,C 180,E1 13310.944,E2 13310.944} C_VEL
LIN {X 0,Y 336.985,Z 514.268,A -85,B 0,C 180,E1 13308.447,E2 13308.447} C_VEL
LIN {X 0,Y 341.01,Z 520.073,A -85,B 0,C 180,E1 13306.002,E2 13306.002} C_VEL
LIN {X 0,Y 346.486,Z 528.291,A -85,B 0,C 180,E1 13303.142,E2 13303.142} C_VEL
LIN {X 0,Y 352.433,Z 537.671,A -85,B 0,C 180,E1 13300.442,E2 13300.442} C_VEL
LIN {X 0,Y 359.308,Z 549.394,A -85,B 0,C 180,E1 13297.677,E2 13297.677} C_VEL
LIN {X 0,Y 360.281,Z 551.418,A -85,B 0,C 180,E1 13297.297,E2 13297.297} C_VEL
LIN {X 0,Y 344.496,Z 760.325,A -85,B 0,C 180,E1 13292.84,E2 13292.84} C_VEL
LIN {X 0,Y 341.525,Z 795.732,A -85,B 0,C 180,E1 13292.024,E2 13292.024} C_VEL
LIN {X 0,Y 338.195,Z 818.567,A -85,B 0,C 180,E1 13291.323,E2 13291.323} C_VEL
LIN {X 0,Y 333.486,Z 841.635,A -85,B 0,C 180,E1 13290.399,E2 13290.399} C_VEL
LIN {X 0,Y 328.295,Z 862.69,A -85,B 0,C 180,E1 13289.299,E2 13289.299} C_VEL
LIN {X 0,Y 322.224,Z 883.543,A -85,B 0,C 180,E1 13287.9,E2 13287.9} C_VEL
LIN {X 0,Y 315.073,Z 905.24,A -85,B 0,C 180,E1 13286.084,E2 13286.084} C_VEL
LIN {X 0,Y 307.774,Z 925.441,A -85,B 0,C 180,E1 13283.991,E2 13283.991} C_VEL
LIN {X 0,Y 300.135,Z 944.771,A -85,B 0,C 180,E1 13281.525,E2 13281.525} C_VEL
LIN {X 0,Y 292.319,Z 963.636,A -85,B 0,C 180,E1 13278.593,E2 13278.593} C_VEL
LIN {X 0,Y 285.054,Z 980.721,A -85,B 0,C 180,E1 13275.402,E2 13275.402} C_VEL
LIN {X 0,Y 278.4,Z 996.164,A -85,B 0,C 180,E1 13271.914,E2 13271.914} C_VEL
LIN {X 0,Y 271.831,Z 1011.943,A -85,B 0,C 180,E1 13267.632,E2 13267.632} C_VEL
LIN {X 0,Y 266.67,Z 1025.311,A -85,B 0,C 180,E1 13263.269,E2 13263.269} C_VEL
LIN {X 0,Y 262.836,Z 1036.388,A -85,B 0,C 180,E1 13258.89,E2 13258.89} C_VEL
LIN {X 0,Y 259.862,Z 1046.982,A -85,B 0,C 180,E1 13253.829,E2 13253.829} C_VEL
LIN {X 0,Y 258.269,Z 1054.903,A -85,B 0,C 180,E1 13249.161,E2 13249.161} C_VEL
LIN {X 0,Y 257.557,Z 1061.203,A -85,B 0,C 180,E1 13244.386,E2 13244.386} C_VEL
LIN {X 0,Y 257.498,Z 1065.294,A -85,B 0,C 180,E1 13240.289,E2 13240.289} C_VEL
LIN {X 0,Y 257.726,Z 1068.224,A -85,B 0,C 180,E1 13236.013,E2 13236.013} C_VEL
LIN {X 0,Y 257.935,Z 1069.53,A -85,B 0,C 180,E1 13231.999,E2 13231.999} C_VEL
LIN {X 0,Y 257.949,Z 1069.59,A -85,B 0,C 180,E1 13228.445,E2 13228.445} C_VEL
LIN {X 0,Y 257.772,Z 1068.495,A -85,B 0,C 180,E1 13224.658,E2 13224.658} C_VEL
LIN {X 0,Y 257.505,Z 1065.88,A -85,B 0,C 180,E1 13220.389,E2 13220.389} C_VEL
LIN {X 0,Y 257.532,Z 1061.708,A -85,B 0,C 180,E1 13216.071,E2 13216.071} C_VEL
LIN {X 0,Y 258.125,Z 1055.857,A -85,B 0,C 180,E1 13211.48,E2 13211.48} C_VEL
LIN {X 0,Y 259.666,Z 1047.809,A -85,B 0,C 180,E1 13206.633,E2 13206.633} C_VEL
LIN {X 0,Y 262.356,Z 1037.976,A -85,B 0,C 180,E1 13201.798,E2 13201.798} C_VEL
LIN {X 0,Y 266.15,Z 1026.661,A -85,B 0,C 180,E1 13197.25,E2 13197.25} C_VEL
LIN {X 0,Y 271.321,Z 1013.157,A -85,B 0,C 180,E1 13192.748,E2 13192.748} C_VEL
LIN {X 0,Y 277.337,Z 998.692,A -85,B 0,C 180,E1 13188.718,E2 13188.718} C_VEL
LIN {X 0,Y 283.791,Z 983.462,A -85,B 0,C 180,E1 13185.199,E2 13185.199} C_VEL
LIN {X 0,Y 291.24,Z 966.069,A -85,B 0,C 180,E1 13181.842,E2 13181.842} C_VEL
LIN {X 0,Y 298.843,Z 947.933,A -85,B 0,C 180,E1 13178.932,E2 13178.932} C_VEL
LIN {X 0,Y 306.325,Z 928.946,A -85,B 0,C 180,E1 13176.445,E2 13176.445} C_VEL
LIN {X 0,Y 314.152,Z 907.63,A -85,B 0,C 180,E1 13174.156,E2 13174.156} C_VEL
LIN {X 0,Y 320.962,Z 887.435,A -85,B 0,C 180,E1 13172.398,E2 13172.398} C_VEL
LIN {X 0,Y 327.064,Z 866.692,A -85,B 0,C 180,E1 13170.961,E2 13170.961} C_VEL
LIN {X 0,Y 332.934,Z 843.628,A -85,B 0,C 180,E1 13169.704,E2 13169.704} C_VEL
LIN {X 0,Y 337.727,Z 820.818,A -85,B 0,C 180,E1 13168.764,E2 13168.764} C_VEL
LIN {X 0,Y 341.192,Z 797.533,A -85,B 0,C 180,E1 13168.038,E2 13168.038} C_VEL
LIN {X 0,Y 343.986,Z 765.822,A -85,B 0,C 180,E1 13167.291,E2 13167.291} C_VEL
LIN {X 0,Y 359.743,Z 556.843,A -85,B 0,C 180,E1 13162.826,E2 13162.826} C_VEL
LIN {X 0,Y 360.161,Z 551.016,A -85,B 0,C 180,E1 13162.698,E2 13162.698} C_VEL
LIN {X 0,Y 353.731,Z 539.984,A -85,B 0,C 180,E1 13160.172,E2 13160.172} C_VEL
LIN {X 0,Y 347.662,Z 530.099,A -85,B 0,C 180,E1 13157.489,E2 13157.489} C_VEL
LIN {X 0,Y 341.436,Z 520.766,A -85,B 0,C 180,E1 13154.326,E2 13154.326} C_VEL
LIN {X 0,Y 337.839,Z 515.632,A -85,B 0,C 180,E1 13152.216,E2 13152.216} C_VEL
LIN {X 0,Y 335.217,Z 511.907,A -85,B 0,C 180,E1 13150.483,E2 13150.483} C_VEL
LIN {X 0,Y 332.008,Z 507.511,A -85,B 0,C 180,E1 13148.049,E2 13148.049} C_VEL
LIN {X 0,Y 328.835,Z 503.153,A -85,B 0,C 180,E1 13145.058,E2 13145.058} C_VEL
LIN {X 0,Y 325.043,Z 497.987,A -85,B 0,C 180,E1 13139.471,E2 13139.471} C_VEL
LIN {X 0,Y 323.853,Z 497.255,A -85,B 0,C 180,E1 13133.974,E2 13133.974} C_VEL
LIN {X 0,Y 324.635,Z 498.119,A -85,B 0,C 180,E1 13130.068,E2 13130.068} C_VEL
LIN {X 0,Y 327.934,Z 503.245,A -85,B 0,C 180,E1 13124.526,E2 13124.526} C_VEL
LIN {X 0,Y 331.189,Z 507.994,A -85,B 0,C 180,E1 13121.244,E2 13121.244} C_VEL
LIN {X 0,Y 334.98,Z 513.676,A -85,B 0,C 180,E1 13118.276,E2 13118.276} C_VEL
LIN {X 0,Y 339.827,Z 520.888,A -85,B 0,C 180,E1 13115.211,E2 13115.211} C_VEL
LIN {X 0,Y 345.447,Z 529.867,A -85,B 0,C 180,E1 13112.225,E2 13112.225} C_VEL
LIN {X 0,Y 351.914,Z 540.635,A -85,B 0,C 180,E1 13109.289,E2 13109.289} C_VEL
LIN {X 0,Y 356.501,Z 549.086,A -85,B 0,C 180,E1 13107.411,E2 13107.411} C_VEL
LIN {X 0,Y 342.968,Z 758.75,A -85,B 0,C 180,E1 13103.343,E2 13103.343} C_VEL
LIN {X 0,Y 340.611,Z 779.658,A -85,B 0,C 180,E1 13102.679,E2 13102.679} C_VEL
LIN {X 0,Y 337.084,Z 800.843,A -85,B 0,C 180,E1 13101.749,E2 13101.749} C_VEL
LIN {X 0,Y 332.925,Z 819.962,A -85,B 0,C 180,E1 13100.655,E2 13100.655} C_VEL
LIN {X 0,Y 327.767,Z 838.733,A -85,B 0,C 180,E1 13099.289,E2 13099.289} C_VEL
LIN {X 0,Y 321.919,Z 856.739,A -85,B 0,C 180,E1 13097.665,E2 13097.665} C_VEL
LIN {X 0,Y 315.443,Z 874.042,A -85,B 0,C 180,E1 13095.755,E2 13095.755} C_VEL
LIN {X 0,Y 308.404,Z 890.521,A -85,B 0,C 180,E1 13093.513,E2 13093.513} C_VEL
LIN {X 0,Y 301.404,Z 905.225,A -85,B 0,C 180,E1 13091.059,E2 13091.059} C_VEL
LIN {X 0,Y 294.17,Z 919.218,A -85,B 0,C 180,E1 13088.215,E2 13088.215} C_VEL
LIN {X 0,Y 287.203,Z 931.84,A -85,B 0,C 180,E1 13085.06,E2 13085.06} C_VEL
LIN {X 0,Y 280.281,Z 943.556,A -85,B 0,C 180,E1 13081.388,E2 13081.388} C_VEL
LIN {X 0,Y 274.387,Z 953.25,A -85,B 0,C 180,E1 13077.567,E2 13077.567} C_VEL
LIN {X 0,Y 269.273,Z 961.597,A -85,B 0,C 180,E1 13073.41,E2 13073.41} C_VEL
LIN {X 0,Y 265.17,Z 968.513,A -85,B 0,C 180,E1 13068.922,E2 13068.922} C_VEL
LIN {X 0,Y 262.086,Z 973.857,A -85,B 0,C 180,E1 13064.132,E2 13064.132} C_VEL
LIN {X 0,Y 260.271,Z 977.343,A -85,B 0,C 180,E1 13059.508,E2 13059.508} C_VEL
LIN {X 0,Y 259.271,Z 979.503,A -85,B 0,C 180,E1 13054.645,E2 13054.645} C_VEL
LIN {X 0,Y 259.003,Z 980.225,A -85,B 0,C 180,E1 13050,E2 13050} C_VEL
LIN {X 0,Y 259.259,Z 979.535,A -85,B 0,C 180,E1 13045.355,E2 13045.355} C_VEL
LIN {X 0,Y 260.252,Z 977.418,A -85,B 0,C 180,E1 13040.491,E2 13040.491} C_VEL
LIN {X 0,Y 262.158,Z 973.756,A -85,B 0,C 180,E1 13035.646,E2 13035.646} C_VEL
LIN {X 0,Y 265.285,Z 968.382,A -85,B 0,C 180,E1 13030.858,E2 13030.858} C_VEL
LIN {X 0,Y 269.427,Z 961.426,A -85,B 0,C 180,E1 13026.372,E2 13026.372} C_VEL
LIN {X 0,Y 274.575,Z 953.026,A -85,B 0,C 180,E1 13022.218,E2 13022.218} C_VEL
LIN {X 0,Y 280.847,Z 942.692,A -85,B 0,C 180,E1 13018.203,E2 13018.203} C_VEL
LIN {X 0,Y 287.463,Z 931.489,A -85,B 0,C 180,E1 13014.733,E2 13014.733} C_VEL
LIN {X 0,Y 294.47,Z 918.825,A -85,B 0,C 180,E1 13011.584,E2 13011.584} C_VEL
LIN {X 0,Y 301.731,Z 904.744,A -85,B 0,C 180,E1 13008.743,E2 13008.743} C_VEL
LIN {X 0,Y 309.165,Z 888.99,A -85,B 0,C 180,E1 13006.154,E2 13006.154} C_VEL
LIN {X 0,Y 316.088,Z 872.735,A -85,B 0,C 180,E1 13003.975,E2 13003.975} C_VEL
LIN {X 0,Y 322.591,Z 855.156,A -85,B 0,C 180,E1 13002.07,E2 13002.07} C_VEL
LIN {X 0,Y 328.464,Z 836.708,A -85,B 0,C 180,E1 13000.446,E2 13000.446} C_VEL
LIN {X 0,Y 332.027,Z 823.787,A -85,B 0,C 180,E1 12999.501,E2 12999.501} C_VEL
LIN {X 0,Y 333.145,Z 817.891,A -85,B 0,C 180,E1 12999.003,E2 12999.003} C_VEL
LIN {X 0,Y 333.738,Z 799.889,A -85,B 0,C 180,E1 12997.077,E2 12997.077} C_VEL
LIN {X 0,Y 334.487,Z 792.726,A -85,B 0,C 180,E1 12996.59,E2 12996.59} C_VEL
LIN {X 0,Y 337.545,Z 772.475,A -85,B 0,C 180,E1 12995.798,E2 12995.798} C_VEL
LIN {X 0,Y 339.494,Z 751.493,A -85,B 0,C 180,E1 12995.226,E2 12995.226} C_VEL
LIN {X 0,Y 352.73,Z 553.209,A -85,B 0,C 180,E1 12991.395,E2 12991.395} C_VEL
LIN {X 0,Y 346.189,Z 541.69,A -85,B 0,C 180,E1 12988.508,E2 12988.508} C_VEL
LIN {X 0,Y 339.967,Z 531.231,A -85,B 0,C 180,E1 12985.29,E2 12985.29} C_VEL
LIN {X 0,Y 335.193,Z 523.691,A -85,B 0,C 180,E1 12982.354,E2 12982.354} C_VEL
LIN {X 0,Y 331.722,Z 518.575,A -85,B 0,C 180,E1 12979.822,E2 12979.822} C_VEL
LIN {X 0,Y 329.112,Z 514.514,A -85,B 0,C 180,E1 12977.504,E2 12977.504} C_VEL
LIN {X 0,Y 326.351,Z 510.341,A -85,B 0,C 180,E1 12974.369,E2 12974.369} C_VEL
LIN {X 0,Y 323.566,Z 505.727,A -85,B 0,C 180,E1 12968.71,E2 12968.71} C_VEL
LIN {X 0,Y 323.359,Z 505.481,A -85,B 0,C 180,E1 12963.369,E2 12963.369} C_VEL
LIN {X 0,Y 324.45,Z 506.416,A -85,B 0,C 180,E1 12960.177,E2 12960.177} C_VEL
LIN {X 0,Y 328.269,Z 511.799,A -85,B 0,C 180,E1 12954.67,E2 12954.67} C_VEL
LIN {X 0,Y 332.01,Z 517.053,A -85,B 0,C 180,E1 12951.253,E2 12951.253} C_VEL
LIN {X 0,Y 335.44,Z 521.976,A -85,B 0,C 180,E1 12948.742,E2 12948.742} C_VEL
LIN {X 0,Y 339.253,Z 527.6,A -85,B 0,C 180,E1 12946.363,E2 12946.363} C_VEL
LIN {X 0,Y 344.931,Z 536.355,A -85,B 0,C 180,E1 12943.324,E2 12943.324} C_VEL
LIN {X 0,Y 350.265,Z 545.104,A -85,B 0,C 180,E1 12940.836,E2 12940.836} C_VEL
LIN {X 0,Y 356.218,Z 555.481,A -85,B 0,C 180,E1 12938.354,E2 12938.354} C_VEL
LIN {X 0,Y 340.828,Z 753.17,A -85,B 0,C 180,E1 12934.138,E2 12934.138} C_VEL
LIN {X 0,Y 337.415,Z 794.042,A -85,B 0,C 180,E1 12933.211,E2 12933.211} C_VEL
LIN {X 0,Y 334.011,Z 817.023,A -85,B 0,C 180,E1 12932.512,E2 12932.512} C_VEL
LIN {X 0,Y 329.3,Z 839.831,A -85,B 0,C 180,E1 12931.616,E2 12931.616} C_VEL
LIN {X 0,Y 323.903,Z 861.247,A -85,B 0,C 180,E1 12930.519,E2 12930.519} C_VEL
LIN {X 0,Y 317.523,Z 882.523,A -85,B 0,C 180,E1 12929.103,E2 12929.103} C_VEL
LIN {X 0,Y 310.142,Z 904.216,A -85,B 0,C 180,E1 12927.292,E2 12927.292} C_VEL
LIN {X 0,Y 302.87,Z 923.664,A -85,B 0,C 180,E1 12925.288,E2 12925.288} C_VEL
LIN {X 0,Y 294.903,Z 943.037,A -85,B 0,C 180,E1 12922.822,E2 12922.822} C_VEL
LIN {X 0,Y 286.48,Z 962.519,A -85,B 0,C 180,E1 12919.784,E2 12919.784} C_VEL
LIN {X 0,Y 278.874,Z 979.585,A -85,B 0,C 180,E1 12916.555,E2 12916.555} C_VEL
LIN {X 0,Y 271.665,Z 995.437,A -85,B 0,C 180,E1 12912.912,E2 12912.912} C_VEL
LIN {X 0,Y 265.071,Z 1010.387,A -85,B 0,C 180,E1 12908.768,E2 12908.768} C_VEL
LIN {X 0,Y 259.718,Z 1023.36,A -85,B 0,C 180,E1 12904.466,E2 12904.466} C_VEL
LIN {X 0,Y 255.415,Z 1034.876,A -85,B 0,C 180,E1 12899.812,E2 12899.812} C_VEL
LIN {X 0,Y 252.28,Z 1045.1,A -85,B 0,C 180,E1 12894.827,E2 12894.827} C_VEL
LIN {X 0,Y 250.563,Z 1052.63,A -85,B 0,C 180,E1 12890.314,E2 12890.314} C_VEL
LIN {X 0,Y 249.665,Z 1059.428,A -85,B 0,C 180,E1 12885.173,E2 12885.173} C_VEL
LIN {X 0,Y 249.553,Z 1063.558,A -85,B 0,C 180,E1 12881.008,E2 12881.008} C_VEL
LIN {X 0,Y 249.777,Z 1066.74,A -85,B 0,C 180,E1 12876.435,E2 12876.435} C_VEL
LIN {X 0,Y 250.029,Z 1068.129,A -85,B 0,C 180,E1 12872.292,E2 12872.292} C_VEL
LIN {X 0,Y 250.066,Z 1068.252,A -85,B 0,C 180,E1 12868.625,E2 12868.625} C_VEL
LIN {X 0,Y 249.893,Z 1067.299,A -85,B 0,C 180,E1 12864.95,E2 12864.95} C_VEL
LIN {X 0,Y 249.602,Z 1064.99,A -85,B 0,C 180,E1 12860.78,E2 12860.78} C_VEL
LIN {X 0,Y 249.585,Z 1060.8,A -85,B 0,C 180,E1 12856.092,E2 12856.092} C_VEL
LIN {X 0,Y 250.077,Z 1055.669,A -85,B 0,C 180,E1 12851.828,E2 12851.828} C_VEL
LIN {X 0,Y 251.658,Z 1047.601,A -85,B 0,C 180,E1 12846.59,E2 12846.59} C_VEL
LIN {X 0,Y 254.318,Z 1038.259,A -85,B 0,C 180,E1 12841.72,E2 12841.72} C_VEL
LIN {X 0,Y 258.294,Z 1026.926,A -85,B 0,C 180,E1 12836.919,E2 12836.919} C_VEL
LIN {X 0,Y 263.546,Z 1013.956,A -85,B 0,C 180,E1 12832.351,E2 12832.351} C_VEL
LIN {X 0,Y 269.456,Z 1000.346,A -85,B 0,C 180,E1 12828.378,E2 12828.378} C_VEL
LIN {X 0,Y 276.513,Z 984.577,A -85,B 0,C 180,E1 12824.546,E2 12824.546} C_VEL
LIN {X 0,Y 284.142,Z 967.733,A -85,B 0,C 180,E1 12821.145,E2 12821.145} C_VEL
LIN {X 0,Y 291.951,Z 949.872,A -85,B 0,C 180,E1 12818.188,E2 12818.188} C_VEL
LIN {X 0,Y 299.943,Z 930.677,A -85,B 0,C 180,E1 12815.572,E2 12815.572} C_VEL
LIN {X 0,Y 307.647,Z 910.891,A -85,B 0,C 180,E1 12813.357,E2 12813.357} C_VEL
LIN {X 0,Y 314.885,Z 890.288,A -85,B 0,C 180,E1 12811.507,E2 12811.507} C_VEL
LIN {X 0,Y 321.494,Z 869.176,A -85,B 0,C 180,E1 12809.985,E2 12809.985} C_VEL
LIN {X 0,Y 327.512,Z 847.016,A -85,B 0,C 180,E1 12808.723,E2 12808.723} C_VEL
LIN {X 0,Y 332.528,Z 824.354,A -85,B 0,C 180,E1 12807.761,E2 12807.761} C_VEL
LIN {X 0,Y 336.46,Z 800.471,A -85,B 0,C 180,E1 12806.982,E2 12806.982} C_VEL
LIN {X 0,Y 338.989,Z 776.041,A -85,B 0,C 180,E1 12806.372,E2 12806.372} C_VEL
LIN {X 0,Y 355.027,Z 569.246,A -85,B 0,C 180,E1 12801.947,E2 12801.947} C_VEL
LIN {X 0,Y 356.025,Z 555.271,A -85,B 0,C 180,E1 12801.626,E2 12801.626} C_VEL
LIN {X 0,Y 348.588,Z 542.297,A -85,B 0,C 180,E1 12798.478,E2 12798.478} C_VEL
LIN {X 0,Y 342.221,Z 532.173,A -85,B 0,C 180,E1 12795.37,E2 12795.37} C_VEL
LIN {X 0,Y 336.801,Z 524.046,A -85,B 0,C 180,E1 12792.254,E2 12792.254} C_VEL
LIN {X 0,Y 333.599,Z 519.421,A -85,B 0,C 180,E1 12790.098,E2 12790.098} C_VEL
LIN {X 0,Y 330.595,Z 515.176,A -85,B 0,C 180,E1 12787.734,E2 12787.734} C_VEL
LIN {X 0,Y 327.513,Z 510.877,A -85,B 0,C 180,E1 12784.728,E2 12784.728} C_VEL
LIN {X 0,Y 323.98,Z 505.883,A -85,B 0,C 180,E1 12779.292,E2 12779.292} C_VEL
LIN {X 0,Y 322.891,Z 505.206,A -85,B 0,C 180,E1 12773.777,E2 12773.777} C_VEL
LIN {X 0,Y 323.616,Z 506.016,A -85,B 0,C 180,E1 12770.216,E2 12770.216} C_VEL
LIN {X 0,Y 326.76,Z 511.099,A -85,B 0,C 180,E1 12764.742,E2 12764.742} C_VEL
LIN {X 0,Y 329.847,Z 515.741,A -85,B 0,C 180,E1 12761.532,E2 12761.532} C_VEL
LIN {X 0,Y 333.448,Z 521.261,A -85,B 0,C 180,E1 12758.634,E2 12758.634} C_VEL
LIN {X 0,Y 338.05,Z 528.303,A -85,B 0,C 180,E1 12755.631,E2 12755.631} C_VEL
LIN {X 0,Y 343.466,Z 537.179,A -85,B 0,C 180,E1 12752.662,E2 12752.662} C_VEL
LIN {X 0,Y 349.79,Z 548.018,A -85,B 0,C 180,E1 12749.7,E2 12749.7} C_VEL
LIN {X 0,Y 352.612,Z 553.467,A -85,B 0,C 180,E1 12748.488,E2 12748.488} C_VEL
LIN {X 0,Y 338.778,Z 759.342,A -85,B 0,C 180,E1 12744.484,E2 12744.484} C_VEL
LIN {X 0,Y 336.331,Z 780.371,A -85,B 0,C 180,E1 12743.817,E2 12743.817} C_VEL
LIN {X 0,Y 332.636,Z 801.838,A -85,B 0,C 180,E1 12742.874,E2 12742.874} C_VEL
LIN {X 0,Y 328.347,Z 820.924,A -85,B 0,C 180,E1 12741.781,E2 12741.781} C_VEL
LIN {X 0,Y 323.039,Z 839.656,A -85,B 0,C 180,E1 12740.417,E2 12740.417} C_VEL
LIN {X 0,Y 316.711,Z 858.48,A -85,B 0,C 180,E1 12738.71,E2 12738.71} C_VEL
LIN {X 0,Y 310.027,Z 875.657,A -85,B 0,C 180,E1 12736.792,E2 12736.792} C_VEL
LIN {X 0,Y 302.829,Z 891.947,A -85,B 0,C 180,E1 12734.557,E2 12734.557} C_VEL
LIN {X 0,Y 295.518,Z 906.725,A -85,B 0,C 180,E1 12732.061,E2 12732.061} C_VEL
LIN {X 0,Y 287.567,Z 921.457,A -85,B 0,C 180,E1 12729.001,E2 12729.001} C_VEL
LIN {X 0,Y 280.367,Z 933.925,A -85,B 0,C 180,E1 12725.794,E2 12725.794} C_VEL
LIN {X 0,Y 273.212,Z 945.554,A -85,B 0,C 180,E1 12722.05,E2 12722.05} C_VEL
LIN {X 0,Y 267.095,Z 955.113,A -85,B 0,C 180,E1 12718.143,E2 12718.143} C_VEL
LIN {X 0,Y 261.541,Z 963.699,A -85,B 0,C 180,E1 12713.667,E2 12713.667} C_VEL
LIN {X 0,Y 257.326,Z 970.417,A -85,B 0,C 180,E1 12709.05,E2 12709.05} C_VEL
LIN {X 0,Y 254.188,Z 975.66,A -85,B 0,C 180,E1 12704.116,E2 12704.116} C_VEL
LIN {X 0,Y 252.288,Z 979.119,A -85,B 0,C 180,E1 12699.121,E2 12699.121} C_VEL
LIN {X 0,Y 251.347,Z 980.982,A -85,B 0,C 180,E1 12694.335,E2 12694.335} C_VEL
LIN {X 0,Y 251.113,Z 981.562,A -85,B 0,C 180,E1 12689.544,E2 12689.544} C_VEL
LIN {X 0,Y 251.461,Z 980.79,A -85,B 0,C 180,E1 12684.753,E2 12684.753} C_VEL
LIN {X 0,Y 252.526,Z 978.652,A -85,B 0,C 180,E1 12679.967,E2 12679.967} C_VEL
LIN {X 0,Y 254.61,Z 974.911,A -85,B 0,C 180,E1 12674.978,E2 12674.978} C_VEL
LIN {X 0,Y 257.805,Z 969.761,A -85,B 0,C 180,E1 12670.28,E2 12670.28} C_VEL
LIN {X 0,Y 262.181,Z 962.808,A -85,B 0,C 180,E1 12665.677,E2 12665.677} C_VEL
LIN {X 0,Y 267.627,Z 954.359,A -85,B 0,C 180,E1 12661.399,E2 12661.399} C_VEL
LIN {X 0,Y 274.154,Z 944.102,A -85,B 0,C 180,E1 12657.332,E2 12657.332} C_VEL
LIN {X 0,Y 281.051,Z 932.928,A -85,B 0,C 180,E1 12653.803,E2 12653.803} C_VEL
LIN {X 0,Y 288.332,Z 920.275,A -85,B 0,C 180,E1 12650.61,E2 12650.61} C_VEL
LIN {X 0,Y 295.863,Z 906.241,A -85,B 0,C 180,E1 12647.738,E2 12647.738} C_VEL
LIN {X 0,Y 303.453,Z 890.778,A -85,B 0,C 180,E1 12645.161,E2 12645.161} C_VEL
LIN {X 0,Y 310.572,Z 874.66,A -85,B 0,C 180,E1 12642.973,E2 12642.973} C_VEL
LIN {X 0,Y 317.123,Z 857.664,A -85,B 0,C 180,E1 12641.101,E2 12641.101} C_VEL
LIN {X 0,Y 323.462,Z 838.62,A -85,B 0,C 180,E1 12639.395,E2 12639.395} C_VEL
LIN {X 0,Y 328.782,Z 819.629,A -85,B 0,C 180,E1 12638.033,E2 12638.033} C_VEL
LIN {X 0,Y 333.101,Z 800.195,A -85,B 0,C 180,E1 12636.939,E2 12636.939} C_VEL
LIN {X 0,Y 334.487,Z 792.726,A -85,B 0,C 180,E1 12636.59,E2 12636.59} C_VEL
LIN {X 0,Y 335.226,Z 785.466,A -85,B 0,C 180,E1 12636.123,E2 12636.123} C_VEL
LIN {X 0,Y 334.635,Z 767.473,A -85,B 0,C 180,E1 12634.591,E2 12634.591} C_VEL
LIN {X 0,Y 334.852,Z 760.012,A -85,B 0,C 180,E1 12634.246,E2 12634.246} C_VEL
LIN {X 0,Y 348.934,Z 557.685,A -85,B 0,C 180,E1 12630.287,E2 12630.287} C_VEL
LIN {X 0,Y 343.274,Z 547.486,A -85,B 0,C 180,E1 12627.636,E2 12627.636} C_VEL
LIN {X 0,Y 337.806,Z 538.095,A -85,B 0,C 180,E1 12624.667,E2 12624.667} C_VEL
LIN {X 0,Y 333.392,Z 530.931,A -85,B 0,C 180,E1 12621.832,E2 12621.832} C_VEL
LIN {X 0,Y 330.153,Z 526.003,A -85,B 0,C 180,E1 12619.368,E2 12619.368} C_VEL
LIN {X 0,Y 327.722,Z 522.125,A -85,B 0,C 180,E1 12617.123,E2 12617.123} C_VEL
LIN {X 0,Y 325.138,Z 518.1,A -85,B 0,C 180,E1 12614.061,E2 12614.061} C_VEL
LIN {X 0,Y 322.565,Z 513.635,A -85,B 0,C 180,E1 12608.557,E2 12608.557} C_VEL
LIN {X 0,Y 322.438,Z 513.456,A -85,B 0,C 180,E1 12603.131,E2 12603.131} C_VEL
LIN {X 0,Y 323.389,Z 514.29,A -85,B 0,C 180,E1 12600.355,E2 12600.355} C_VEL
LIN {X 0,Y 327.009,Z 519.598,A -85,B 0,C 180,E1 12594.913,E2 12594.913} C_VEL
LIN {X 0,Y 330.562,Z 524.728,A -85,B 0,C 180,E1 12591.565,E2 12591.565} C_VEL
LIN {X 0,Y 333.793,Z 529.488,A -85,B 0,C 180,E1 12589.123,E2 12589.123} C_VEL
LIN {X 0,Y 337.784,Z 535.534,A -85,B 0,C 180,E1 12586.564,E2 12586.564} C_VEL
LIN {X 0,Y 343.618,Z 544.763,A -85,B 0,C 180,E1 12583.389,E2 12583.389} C_VEL
LIN {X 0,Y 349.841,Z 555.529,A -85,B 0,C 180,E1 12580.465,E2 12580.465} C_VEL
LIN {X 0,Y 352.263,Z 560.114,A -85,B 0,C 180,E1 12579.414,E2 12579.414} C_VEL
LIN {X 0,Y 335.399,Z 770.866,A -85,B 0,C 180,E1 12574.924,E2 12574.924} C_VEL
LIN {X 0,Y 332.654,Z 798.257,A -85,B 0,C 180,E1 12574.261,E2 12574.261} C_VEL
LIN {X 0,Y 328.925,Z 821.256,A -85,B 0,C 180,E1 12573.534,E2 12573.534} C_VEL
LIN {X 0,Y 323.974,Z 843.397,A -85,B 0,C 180,E1 12572.623,E2 12572.623} C_VEL
LIN {X 0,Y 317.971,Z 865.434,A -85,B 0,C 180,E1 12571.427,E2 12571.427} C_VEL
LIN {X 0,Y 311.621,Z 885.698,A -85,B 0,C 180,E1 12570.034,E2 12570.034} C_VEL
LIN {X 0,Y 304.341,Z 905.869,A -85,B 0,C 180,E1 12568.289,E2 12568.289} C_VEL
LIN {X 0,Y 296.007,Z 926.884,A -85,B 0,C 180,E1 12566.032,E2 12566.032} C_VEL
LIN {X 0,Y 287.893,Z 945.831,A -85,B 0,C 180,E1 12563.532,E2 12563.532} C_VEL
LIN {X 0,Y 279.594,Z 963.956,A -85,B 0,C 180,E1 12560.574,E2 12560.574} C_VEL
LIN {X 0,Y 271.425,Z 981.267,A -85,B 0,C 180,E1 12557.144,E2 12557.144} C_VEL
LIN {X 0,Y 263.855,Z 997.255,A -85,B 0,C 180,E1 12553.306,E2 12553.306} C_VEL
LIN {X 0,Y 257.114,Z 1011.726,A -85,B 0,C 180,E1 12549.049,E2 12549.049} C_VEL
LIN {X 0,Y 251.412,Z 1024.839,A -85,B 0,C 180,E1 12544.384,E2 12544.384} C_VEL
LIN {X 0,Y 247.103,Z 1036.12,A -85,B 0,C 180,E1 12539.548,E2 12539.548} C_VEL
LIN {X 0,Y 244.068,Z 1045.723,A -85,B 0,C 180,E1 12534.442,E2 12534.442} C_VEL
LIN {X 0,Y 242.277,Z 1053.925,A -85,B 0,C 180,E1 12529.028,E2 12529.028} C_VEL
LIN {X 0,Y 241.66,Z 1059.389,A -85,B 0,C 180,E1 12524.374,E2 12524.374} C_VEL
LIN {X 0,Y 241.672,Z 1063.604,A -85,B 0,C 180,E1 12519.526,E2 12519.526} C_VEL
LIN {X 0,Y 241.987,Z 1065.928,A -85,B 0,C 180,E1 12515.215,E2 12515.215} C_VEL
LIN {X 0,Y 242.181,Z 1066.888,A -85,B 0,C 180,E1 12511.419,E2 12511.419} C_VEL
LIN {X 0,Y 242.138,Z 1066.76,A -85,B 0,C 180,E1 12507.633,E2 12507.633} C_VEL
LIN {X 0,Y 241.859,Z 1065.353,A -85,B 0,C 180,E1 12503.353,E2 12503.353} C_VEL
LIN {X 0,Y 241.625,Z 1062.228,A -85,B 0,C 180,E1 12498.726,E2 12498.726} C_VEL
LIN {X 0,Y 241.752,Z 1058.081,A -85,B 0,C 180,E1 12494.405,E2 12494.405} C_VEL
LIN {X 0,Y 242.689,Z 1051.517,A -85,B 0,C 180,E1 12489.248,E2 12489.248} C_VEL
LIN {X 0,Y 244.531,Z 1043.995,A -85,B 0,C 180,E1 12484.574,E2 12484.574} C_VEL
LIN {X 0,Y 247.868,Z 1033.873,A -85,B 0,C 180,E1 12479.451,E2 12479.451} C_VEL
LIN {X 0,Y 252.426,Z 1022.405,A -85,B 0,C 180,E1 12474.668,E2 12474.668} C_VEL
LIN {X 0,Y 258.083,Z 1009.499,A -85,B 0,C 180,E1 12470.265,E2 12470.265} C_VEL
LIN {X 0,Y 265.021,Z 994.627,A -85,B 0,C 180,E1 12466.037,E2 12466.037} C_VEL
LIN {X 0,Y 272.567,Z 978.833,A -85,B 0,C 180,E1 12462.339,E2 12462.339} C_VEL
LIN {X 0,Y 280.605,Z 961.626,A -85,B 0,C 180,E1 12459.032,E2 12459.032} C_VEL
LIN {X 0,Y 288.855,Z 943.422,A -85,B 0,C 180,E1 12456.146,E2 12456.146} C_VEL
LIN {X 0,Y 296.892,Z 924.61,A -85,B 0,C 180,E1 12453.712,E2 12453.712} C_VEL
LIN {X 0,Y 304.692,Z 904.7,A -85,B 0,C 180,E1 12451.617,E2 12451.617} C_VEL
LIN {X 0,Y 311.892,Z 884.573,A -85,B 0,C 180,E1 12449.897,E2 12449.897} C_VEL
LIN {X 0,Y 318.11,Z 864.641,A -85,B 0,C 180,E1 12448.538,E2 12448.538} C_VEL
LIN {X 0,Y 324.159,Z 842.185,A -85,B 0,C 180,E1 12447.335,E2 12447.335} C_VEL
LIN {X 0,Y 329.152,Z 819.627,A -85,B 0,C 180,E1 12446.418,E2 12446.418} C_VEL
LIN {X 0,Y 332.809,Z 796.267,A -85,B 0,C 180,E1 12445.696,E2 12445.696} C_VEL
LIN {X 0,Y 335.78,Z 764.567,A -85,B 0,C 180,E1 12444.95,E2 12444.95} C_VEL
LIN {X 0,Y 352.156,Z 559.753,A -85,B 0,C 180,E1 12440.586,E2 12440.586} C_VEL
LIN {X 0,Y 344.902,Z 547.089,A -85,B 0,C 180,E1 12437.329,E2 12437.329} C_VEL
LIN {X 0,Y 338.466,Z 536.598,A -85,B 0,C 180,E1 12433.931,E2 12433.931} C_VEL
LIN {X 0,Y 334.107,Z 530.086,A -85,B 0,C 180,E1 12431.216,E2 12431.216} C_VEL
LIN {X 0,Y 331.765,Z 526.636,A -85,B 0,C 180,E1 12429.541,E2 12429.541} C_VEL
LIN {X 0,Y 329.092,Z 522.721,A -85,B 0,C 180,E1 12427.331,E2 12427.331} C_VEL
LIN {X 0,Y 326.201,Z 518.602,A -85,B 0,C 180,E1 12424.394,E2 12424.394} C_VEL
LIN {X 0,Y 322.985,Z 513.818,A -85,B 0,C 180,E1 12419.247,E2 12419.247} C_VEL
LIN {X 0,Y 321.921,Z 513.15,A -85,B 0,C 180,E1 12413.759,E2 12413.759} C_VEL
LIN {X 0,Y 322.599,Z 513.914,A -85,B 0,C 180,E1 12410.365,E2 12410.365} C_VEL
LIN {X 0,Y 325.532,Z 518.813,A -85,B 0,C 180,E1 12405.048,E2 12405.048} C_VEL
LIN {X 0,Y 328.529,Z 523.486,A -85,B 0,C 180,E1 12401.823,E2 12401.823} C_VEL
LIN {X 0,Y 331.931,Z 528.843,A -85,B 0,C 180,E1 12398.994,E2 12398.994} C_VEL
LIN {X 0,Y 336.291,Z 535.717,A -85,B 0,C 180,E1 12396.056,E2 12396.056} C_VEL
LIN {X 0,Y 341.811,Z 544.997,A -85,B 0,C 180,E1 12392.943,E2 12392.943} C_VEL
LIN {X 0,Y 347.851,Z 555.778,A -85,B 0,C 180,E1 12390.037,E2 12390.037} C_VEL
LIN {X 0,Y 348.837,Z 557.901,A -85,B 0,C 180,E1 12389.587,E2 12389.587} C_VEL
LIN {X 0,Y 334.722,Z 759.991,A -85,B 0,C 180,E1 12385.652,E2 12385.652} C_VEL
LIN {X 0,Y 332.206,Z 780.942,A -85,B 0,C 180,E1 12384.988,E2 12384.988} C_VEL
LIN {X 0,Y 328.475,Z 802.105,A -85,B 0,C 180,E1 12384.066,E2 12384.066} C_VEL
LIN {X 0,Y 323.899,Z 821.88,A -85,B 0,C 180,E1 12382.938,E2 12382.938} C_VEL
LIN {X 0,Y 318.273,Z 841.112,A -85,B 0,C 180,E1 12381.536,E2 12381.536} C_VEL
LIN {X 0,Y 312.029,Z 859.096,A -85,B 0,C 180,E1 12379.903,E2 12379.903} C_VEL
LIN {X 0,Y 305,Z 876.633,A -85,B 0,C 180,E1 12377.947,E2 12377.947} C_VEL
LIN {X 0,Y 297.554,Z 892.943,A -85,B 0,C 180,E1 12375.704,E2 12375.704} C_VEL
LIN {X 0,Y 290.233,Z 907.277,A -85,B 0,C 180,E1 12373.28,E2 12373.28} C_VEL
LIN {X 0,Y 282.418,Z 921.338,A -85,B 0,C 180,E1 12370.383,E2 12370.383} C_VEL
LIN {X 0,Y 274.842,Z 934.015,A -85,B 0,C 180,E1 12367.15,E2 12367.15} C_VEL
LIN {X 0,Y 267.64,Z 945.223,A -85,B 0,C 180,E1 12363.567,E2 12363.567} C_VEL
LIN {X 0,Y 260.752,Z 955.582,A -85,B 0,C 180,E1 12359.395,E2 12359.395} C_VEL
LIN {X 0,Y 255.057,Z 964.006,A -85,B 0,C 180,E1 12355.048,E2 12355.048} C_VEL
LIN {X 0,Y 250.411,Z 970.99,A -85,B 0,C 180,E1 12350.327,E2 12350.327} C_VEL
LIN {X 0,Y 246.882,Z 976.391,A -85,B 0,C 180,E1 12345.263,E2 12345.263} C_VEL
LIN {X 0,Y 244.69,Z 980.084,A -85,B 0,C 180,E1 12340.12,E2 12340.12} C_VEL
LIN {X 0,Y 243.547,Z 982.236,A -85,B 0,C 180,E1 12334.946,E2 12334.946} C_VEL
LIN {X 0,Y 243.237,Z 982.956,A -85,B 0,C 180,E1 12330,E2 12330} C_VEL
LIN {X 0,Y 243.535,Z 982.267,A -85,B 0,C 180,E1 12325.054,E2 12325.054} C_VEL
LIN {X 0,Y 244.669,Z 980.158,A -85,B 0,C 180,E1 12319.879,E2 12319.879} C_VEL
LIN {X 0,Y 246.718,Z 976.726,A -85,B 0,C 180,E1 12314.967,E2 12314.967} C_VEL
LIN {X 0,Y 250.162,Z 971.405,A -85,B 0,C 180,E1 12309.896,E2 12309.896} C_VEL
LIN {X 0,Y 254.721,Z 964.55,A -85,B 0,C 180,E1 12305.165,E2 12305.165} C_VEL
LIN {X 0,Y 260.654,Z 955.814,A -85,B 0,C 180,E1 12300.593,E2 12300.593} C_VEL
LIN {X 0,Y 267.363,Z 945.771,A -85,B 0,C 180,E1 12296.508,E2 12296.508} C_VEL
LIN {X 0,Y 274.717,Z 934.36,A -85,B 0,C 180,E1 12292.83,E2 12292.83} C_VEL
LIN {X 0,Y 282.282,Z 921.723,A -85,B 0,C 180,E1 12289.594,E2 12289.594} C_VEL
LIN {X 0,Y 290.343,Z 907.258,A -85,B 0,C 180,E1 12286.605,E2 12286.605} C_VEL
LIN {X 0,Y 298.207,Z 891.764,A -85,B 0,C 180,E1 12284.011,E2 12284.011} C_VEL
LIN {X 0,Y 305.703,Z 875.329,A -85,B 0,C 180,E1 12281.779,E2 12281.779} C_VEL
LIN {X 0,Y 312.628,Z 857.831,A -85,B 0,C 180,E1 12279.863,E2 12279.863} C_VEL
LIN {X 0,Y 318.872,Z 839.556,A -85,B 0,C 180,E1 12278.235,E2 12278.235} C_VEL
LIN {X 0,Y 324.355,Z 820.578,A -85,B 0,C 180,E1 12276.875,E2 12276.875} C_VEL
LIN {X 0,Y 328.789,Z 801.242,A -85,B 0,C 180,E1 12275.787,E2 12275.787} C_VEL
LIN {X 0,Y 332.405,Z 780.474,A -85,B 0,C 180,E1 12274.892,E2 12274.892} C_VEL
LIN {X 0,Y 334.852,Z 760.012,A -85,B 0,C 180,E1 12274.246,E2 12274.246} C_VEL
LIN {X 0,Y 334.993,Z 752.477,A -85,B 0,C 180,E1 12273.924,E2 12273.924} C_VEL
LIN {X 0,Y 333.336,Z 732.823,A -85,B 0,C 180,E1 12272.575,E2 12272.575} C_VEL
LIN {X 0,Y 333.42,Z 726.324,A -85,B 0,C 180,E1 12272.333,E2 12272.333} C_VEL
LIN {X 0,Y 345.294,Z 562.106,A -85,B 0,C 180,E1 12269.157,E2 12269.157} C_VEL
LIN {X 0,Y 339.535,Z 551.643,A -85,B 0,C 180,E1 12266.261,E2 12266.261} C_VEL
LIN {X 0,Y 334.564,Z 543.03,A -85,B 0,C 180,E1 12263.328,E2 12263.328} C_VEL
LIN {X 0,Y 330.088,Z 535.7,A -85,B 0,C 180,E1 12260.137,E2 12260.137} C_VEL
LIN {X 0,Y 326.434,Z 529.84,A -85,B 0,C 180,E1 12256.826,E2 12256.826} C_VEL
LIN {X 0,Y 323.936,Z 525.858,A -85,B 0,C 180,E1 12253.749,E2 12253.749} C_VEL
LIN {X 0,Y 321.554,Z 521.543,A -85,B 0,C 180,E1 12248.404,E2 12248.404} C_VEL
LIN {X 0,Y 321.49,Z 521.414,A -85,B 0,C 180,E1 12243.031,E2 12243.031} C_VEL
LIN {X 0,Y 322.321,Z 522.164,A -85,B 0,C 180,E1 12240.534,E2 12240.534} C_VEL
LIN {X 0,Y 325.766,Z 527.397,A -85,B 0,C 180,E1 12235.159,E2 12235.159} C_VEL
LIN {X 0,Y 329.124,Z 532.402,A -85,B 0,C 180,E1 12231.88,E2 12231.88} C_VEL
LIN {X 0,Y 332.277,Z 537.193,A -85,B 0,C 180,E1 12229.424,E2 12229.424} C_VEL
LIN {X 0,Y 336.664,Z 543.946,A -85,B 0,C 180,E1 12226.562,E2 12226.562} C_VEL
LIN {X 0,Y 343.465,Z 555.323,A -85,B 0,C 180,E1 12222.858,E2 12222.858} C_VEL
LIN {X 0,Y 348.436,Z 564.631,A -85,B 0,C 180,E1 12220.505,E2 12220.505} C_VEL
LIN {X 0,Y 331.189,Z 774.159,A -85,B 0,C 180,E1 12216.052,E2 12216.052} C_VEL
LIN {X 0,Y 328.54,Z 798.648,A -85,B 0,C 180,E1 12215.448,E2 12215.448} C_VEL
LIN {X 0,Y 324.53,Z 822.136,A -85,B 0,C 180,E1 12214.698,E2 12214.698} C_VEL
LIN {X 0,Y 319.545,Z 843.734,A -85,B 0,C 180,E1 12213.809,E2 12213.809} C_VEL
LIN {X 0,Y 313.512,Z 865.089,A -85,B 0,C 180,E1 12212.649,E2 12212.649} C_VEL
LIN {X 0,Y 306.829,Z 885.653,A -85,B 0,C 180,E1 12211.234,E2 12211.234} C_VEL
LIN {X 0,Y 299.302,Z 905.81,A -85,B 0,C 180,E1 12209.485,E2 12209.485} C_VEL
LIN {X 0,Y 291.028,Z 925.876,A -85,B 0,C 180,E1 12207.323,E2 12207.323} C_VEL
LIN {X 0,Y 282.588,Z 944.822,A -85,B 0,C 180,E1 12204.819,E2 12204.819} C_VEL
LIN {X 0,Y 273.966,Z 962.861,A -85,B 0,C 180,E1 12201.859,E2 12201.859} C_VEL
LIN {X 0,Y 265.187,Z 980.6,A -85,B 0,C 180,E1 12198.292,E2 12198.292} C_VEL
LIN {X 0,Y 257.653,Z 995.687,A -85,B 0,C 180,E1 12194.62,E2 12194.62} C_VEL
LIN {X 0,Y 250.49,Z 1010.173,A -85,B 0,C 180,E1 12190.289,E2 12190.289} C_VEL
LIN {X 0,Y 244.346,Z 1023.404,A -85,B 0,C 180,E1 12185.483,E2 12185.483} C_VEL
LIN {X 0,Y 239.757,Z 1034.551,A -85,B 0,C 180,E1 12180.583,E2 12180.583} C_VEL
LIN {X 0,Y 236.539,Z 1043.819,A -85,B 0,C 180,E1 12175.541,E2 12175.541} C_VEL
LIN {X 0,Y 234.583,Z 1051.676,A -85,B 0,C 180,E1 12170.334,E2 12170.334} C_VEL
LIN {X 0,Y 233.779,Z 1057.447,A -85,B 0,C 180,E1 12165.377,E2 12165.377} C_VEL
LIN {X 0,Y 233.707,Z 1061.689,A -85,B 0,C 180,E1 12160.601,E2 12160.601} C_VEL
LIN {X 0,Y 234.038,Z 1064.368,A -85,B 0,C 180,E1 12155.885,E2 12155.885} C_VEL
LIN {X 0,Y 234.28,Z 1065.461,A -85,B 0,C 180,E1 12151.957,E2 12151.957} C_VEL
LIN {X 0,Y 234.291,Z 1065.491,A -85,B 0,C 180,E1 12148.288,E2 12148.288} C_VEL
LIN {X 0,Y 234.07,Z 1064.458,A -85,B 0,C 180,E1 12144.362,E2 12144.362} C_VEL
LIN {X 0,Y 233.717,Z 1061.878,A -85,B 0,C 180,E1 12139.649,E2 12139.649} C_VEL
LIN {X 0,Y 233.76,Z 1057.692,A -85,B 0,C 180,E1 12134.875,E2 12134.875} C_VEL
LIN {X 0,Y 234.495,Z 1052.143,A -85,B 0,C 180,E1 12130.055,E2 12130.055} C_VEL
LIN {X 0,Y 236.417,Z 1044.215,A -85,B 0,C 180,E1 12124.713,E2 12124.713} C_VEL
LIN {X 0,Y 239.564,Z 1035.022,A -85,B 0,C 180,E1 12119.667,E2 12119.667} C_VEL
LIN {X 0,Y 244.118,Z 1023.871,A -85,B 0,C 180,E1 12114.724,E2 12114.724} C_VEL
LIN {X 0,Y 250.149,Z 1010.837,A -85,B 0,C 180,E1 12109.944,E2 12109.944} C_VEL
LIN {X 0,Y 257.066,Z 996.747,A -85,B 0,C 180,E1 12105.697,E2 12105.697} C_VEL
LIN {X 0,Y 264.942,Z 980.976,A -85,B 0,C 180,E1 12101.811,E2 12101.811} C_VEL
LIN {X 0,Y 273.43,Z 963.851,A -85,B 0,C 180,E1 12098.337,E2 12098.337} C_VEL
LIN {X 0,Y 281.997,Z 945.893,A -85,B 0,C 180,E1 12095.363,E2 12095.363} C_VEL
LIN {X 0,Y 290.581,Z 926.696,A -85,B 0,C 180,E1 12092.793,E2 12092.793} C_VEL
LIN {X 0,Y 299.244,Z 905.708,A -85,B 0,C 180,E1 12090.522,E2 12090.522} C_VEL
LIN {X 0,Y 306.818,Z 885.415,A -85,B 0,C 180,E1 12088.762,E2 12088.762} C_VEL
LIN {X 0,Y 313.574,Z 864.541,A -85,B 0,C 180,E1 12087.332,E2 12087.332} C_VEL
LIN {X 0,Y 319.885,Z 841.888,A -85,B 0,C 180,E1 12086.122,E2 12086.122} C_VEL
LIN {X 0,Y 324.989,Z 819.452,A -85,B 0,C 180,E1 12085.215,E2 12085.215} C_VEL
LIN {X 0,Y 328.744,Z 796.291,A -85,B 0,C 180,E1 12084.499,E2 12084.499} C_VEL
LIN {X 0,Y 331.773,Z 765.394,A -85,B 0,C 180,E1 12083.769,E2 12083.769} C_VEL
LIN {X 0,Y 348.32,Z 564.35,A -85,B 0,C 180,E1 12079.5,E2 12079.5} C_VEL
LIN {X 0,Y 342.361,Z 553.646,A -85,B 0,C 180,E1 12076.674,E2 12076.674} C_VEL
LIN {X 0,Y 336.426,Z 543.712,A -85,B 0,C 180,E1 12073.403,E2 12073.403} C_VEL
LIN {X 0,Y 331.2,Z 535.453,A -85,B 0,C 180,E1 12069.908,E2 12069.908} C_VEL
LIN {X 0,Y 327.605,Z 530.265,A -85,B 0,C 180,E1 12066.924,E2 12066.924} C_VEL
LIN {X 0,Y 325.051,Z 526.466,A -85,B 0,C 180,E1 12064.233,E2 12064.233} C_VEL
LIN {X 0,Y 321.95,Z 521.729,A -85,B 0,C 180,E1 12059.11,E2 12059.11} C_VEL
LIN {X 0,Y 320.952,Z 521.093,A -85,B 0,C 180,E1 12053.74,E2 12053.74} C_VEL
LIN {X 0,Y 321.576,Z 521.811,A -85,B 0,C 180,E1 12050.514,E2 12050.514} C_VEL
LIN {X 0,Y 324.371,Z 526.664,A -85,B 0,C 180,E1 12045.267,E2 12045.267} C_VEL
LIN {X 0,Y 327.133,Z 531.058,A -85,B 0,C 180,E1 12042.203,E2 12042.203} C_VEL
LIN {X 0,Y 330.428,Z 536.424,A -85,B 0,C 180,E1 12039.358,E2 12039.358} C_VEL
LIN {X 0,Y 334.61,Z 543.245,A -85,B 0,C 180,E1 12036.442,E2 12036.442} C_VEL
LIN {X 0,Y 340.008,Z 552.552,A -85,B 0,C 180,E1 12033.308,E2 12033.308} C_VEL
LIN {X 0,Y 345.2,Z 562.259,A -85,B 0,C 180,E1 12030.711,E2 12030.711} C_VEL
LIN {X 0,Y 330.809,Z 760.62,A -85,B 0,C 180,E1 12026.849,E2 12026.849} C_VEL
LIN {X 0,Y 328.203,Z 781.645,A -85,B 0,C 180,E1 12026.185,E2 12026.185} C_VEL
LIN {X 0,Y 324.299,Z 803.092,A -85,B 0,C 180,E1 12025.252,E2 12025.252} C_VEL
LIN {X 0,Y 319.587,Z 822.835,A -85,B 0,C 180,E1 12024.127,E2 12024.127} C_VEL
LIN {X 0,Y 313.676,Z 842.428,A -85,B 0,C 180,E1 12022.699,E2 12022.699} C_VEL
LIN {X 0,Y 307.223,Z 860.391,A -85,B 0,C 180,E1 12021.063,E2 12021.063} C_VEL
LIN {X 0,Y 300.101,Z 877.606,A -85,B 0,C 180,E1 12019.14,E2 12019.14} C_VEL
LIN {X 0,Y 292.402,Z 893.934,A -85,B 0,C 180,E1 12016.892,E2 12016.892} C_VEL
LIN {X 0,Y 284.557,Z 908.773,A -85,B 0,C 180,E1 12014.366,E2 12014.366} C_VEL
LIN {X 0,Y 275.974,Z 923.579,A -85,B 0,C 180,E1 12011.254,E2 12011.254} C_VEL
LIN {X 0,Y 268.149,Z 936.12,A -85,B 0,C 180,E1 12007.97,E2 12007.97} C_VEL
LIN {X 0,Y 260.316,Z 947.803,A -85,B 0,C 180,E1 12004.11,E2 12004.11} C_VEL
LIN {X 0,Y 253.552,Z 957.441,A -85,B 0,C 180,E1 12000.054,E2 12000.054} C_VEL
LIN {X 0,Y 247.362,Z 966.11,A -85,B 0,C 180,E1 11995.37,E2 11995.37} C_VEL
LIN {X 0,Y 242.589,Z 972.908,A -85,B 0,C 180,E1 11990.508,E2 11990.508} C_VEL
LIN {X 0,Y 238.987,Z 978.209,A -85,B 0,C 180,E1 11985.282,E2 11985.282} C_VEL
LIN {X 0,Y 236.76,Z 981.726,A -85,B 0,C 180,E1 11979.971,E2 11979.971} C_VEL
LIN {X 0,Y 235.619,Z 983.715,A -85,B 0,C 180,E1 11974.625,E2 11974.625} C_VEL
LIN {X 0,Y 235.348,Z 984.292,A -85,B 0,C 180,E1 11969.513,E2 11969.513} C_VEL
LIN {X 0,Y 235.749,Z 983.522,A -85,B 0,C 180,E1 11964.402,E2 11964.402} C_VEL
LIN {X 0,Y 236.967,Z 981.392,A -85,B 0,C 180,E1 11959.301,E2 11959.301} C_VEL
LIN {X 0,Y 239.34,Z 977.661,A -85,B 0,C 180,E1 11953.995,E2 11953.995} C_VEL
LIN {X 0,Y 243.131,Z 972.224,A -85,B 0,C 180,E1 11948.783,E2 11948.783} C_VEL
LIN {X 0,Y 248.088,Z 965.211,A -85,B 0,C 180,E1 11943.941,E2 11943.941} C_VEL
LIN {X 0,Y 254.109,Z 956.743,A -85,B 0,C 180,E1 11939.497,E2 11939.497} C_VEL
LIN {X 0,Y 261.363,Z 946.341,A -85,B 0,C 180,E1 11935.249,E2 11935.249} C_VEL
LIN {X 0,Y 268.902,Z 935.088,A -85,B 0,C 180,E1 11931.614,E2 11931.614} C_VEL
LIN {X 0,Y 276.813,Z 922.382,A -85,B 0,C 180,E1 11928.347,E2 11928.347} C_VEL
LIN {X 0,Y 284.96,Z 908.239,A -85,B 0,C 180,E1 11925.421,E2 11925.421} C_VEL
LIN {X 0,Y 293.084,Z 892.748,A -85,B 0,C 180,E1 11922.821,E2 11922.821} C_VEL
LIN {X 0,Y 300.845,Z 876.265,A -85,B 0,C 180,E1 11920.58,E2 11920.58} C_VEL
LIN {X 0,Y 307.979,Z 858.775,A -85,B 0,C 180,E1 11918.667,E2 11918.667} C_VEL
LIN {X 0,Y 314.418,Z 840.493,A -85,B 0,C 180,E1 11917.042,E2 11917.042} C_VEL
LIN {X 0,Y 320.064,Z 821.524,A -85,B 0,C 180,E1 11915.686,E2 11915.686} C_VEL
LIN {X 0,Y 324.791,Z 801.482,A -85,B 0,C 180,E1 11914.564,E2 11914.564} C_VEL
LIN {X 0,Y 328.434,Z 781.023,A -85,B 0,C 180,E1 11913.69,E2 11913.69} C_VEL
LIN {X 0,Y 331.014,Z 759.767,A -85,B 0,C 180,E1 11913.027,E2 11913.027} C_VEL
LIN {X 0,Y 333.42,Z 726.324,A -85,B 0,C 180,E1 11912.333,E2 11912.333} C_VEL
LIN {X 0,Y 333.486,Z 718.756,A -85,B 0,C 180,E1 11912.032,E2 11912.032} C_VEL
LIN {X 0,Y 332.132,Z 699.044,A -85,B 0,C 180,E1 11910.686,E2 11910.686} C_VEL
LIN {X 0,Y 332.29,Z 692.537,A -85,B 0,C 180,E1 11910.445,E2 11910.445} C_VEL
LIN {X 0,Y 341.765,Z 566.689,A -85,B 0,C 180,E1 11908.006,E2 11908.006} C_VEL
LIN {X 0,Y 335.902,Z 555.822,A -85,B 0,C 180,E1 11904.817,E2 11904.817} C_VEL
LIN {X 0,Y 331.251,Z 547.725,A -85,B 0,C 180,E1 11901.794,E2 11901.794} C_VEL
LIN {X 0,Y 327.474,Z 541.453,A -85,B 0,C 180,E1 11898.801,E2 11898.801} C_VEL
LIN {X 0,Y 324.996,Z 537.342,A -85,B 0,C 180,E1 11896.35,E2 11896.35} C_VEL
LIN {X 0,Y 322.865,Z 533.75,A -85,B 0,C 180,E1 11893.613,E2 11893.613} C_VEL
LIN {X 0,Y 320.543,Z 529.453,A -85,B 0,C 180,E1 11888.25,E2 11888.25} C_VEL
LIN {X 0,Y 320.552,Z 529.38,A -85,B 0,C 180,E1 11882.861,E2 11882.861} C_VEL
LIN {X 0,Y 321.256,Z 530.037,A -85,B 0,C 180,E1 11880.714,E2 11880.714} C_VEL
LIN {X 0,Y 324.532,Z 535.196,A -85,B 0,C 180,E1 11875.406,E2 11875.406} C_VEL
LIN {X 0,Y 327.705,Z 540.077,A -85,B 0,C 180,E1 11872.197,E2 11872.197} C_VEL
LIN {X 0,Y 330.655,Z 544.704,A -85,B 0,C 180,E1 11869.812,E2 11869.812} C_VEL
LIN {X 0,Y 334.787,Z 551.274,A -85,B 0,C 180,E1 11867.013,E2 11867.013} C_VEL
LIN {X 0,Y 341.254,Z 562.415,A -85,B 0,C 180,E1 11863.359,E2 11863.359} C_VEL
LIN {X 0,Y 344.728,Z 569.209,A -85,B 0,C 180,E1 11861.618,E2 11861.618} C_VEL
LIN {X 0,Y 327.152,Z 777.009,A -85,B 0,C 180,E1 11857.219,E2 11857.219} C_VEL
LIN {X 0,Y 324.4,Z 800.259,A -85,B 0,C 180,E1 11856.632,E2 11856.632} C_VEL
LIN {X 0,Y 320.051,Z 824.044,A -85,B 0,C 180,E1 11855.857,E2 11855.857} C_VEL
LIN {X 0,Y 314.628,Z 846.349,A -85,B 0,C 180,E1 11854.919,E2 11854.919} C_VEL
LIN {X 0,Y 308.322,Z 867.545,A -85,B 0,C 180,E1 11853.734,E2 11853.734} C_VEL
LIN {X 0,Y 300.749,Z 889.371,A -85,B 0,C 180,E1 11852.171,E2 11852.171} C_VEL
LIN {X 0,Y 292.78,Z 909.704,A -85,B 0,C 180,E1 11850.339,E2 11850.339} C_VEL
LIN {X 0,Y 284.419,Z 928.846,A -85,B 0,C 180,E1 11848.177,E2 11848.177} C_VEL
LIN {X 0,Y 275.28,Z 948.133,A -85,B 0,C 180,E1 11845.486,E2 11845.486} C_VEL
LIN {X 0,Y 266.302,Z 966.099,A -85,B 0,C 180,E1 11842.394,E2 11842.394} C_VEL
LIN {X 0,Y 257.811,Z 982.322,A -85,B 0,C 180,E1 11838.953,E2 11838.953} C_VEL
LIN {X 0,Y 249.47,Z 998.077,A -85,B 0,C 180,E1 11834.862,E2 11834.862} C_VEL
LIN {X 0,Y 242.223,Z 1012.167,A -85,B 0,C 180,E1 11830.397,E2 11830.397} C_VEL
LIN {X 0,Y 236.074,Z 1024.783,A -85,B 0,C 180,E1 11825.468,E2 11825.468} C_VEL
LIN {X 0,Y 231.267,Z 1035.973,A -85,B 0,C 180,E1 11820.1,E2 11820.1} C_VEL
LIN {X 0,Y 228.073,Z 1045.284,A -85,B 0,C 180,E1 11814.612,E2 11814.612} C_VEL
LIN {X 0,Y 226.319,Z 1052.688,A -85,B 0,C 180,E1 11809.017,E2 11809.017} C_VEL
LIN {X 0,Y 225.744,Z 1058.234,A -85,B 0,C 180,E1 11803.577,E2 11803.577} C_VEL
LIN {X 0,Y 225.879,Z 1061.567,A -85,B 0,C 180,E1 11798.913,E2 11798.913} C_VEL
LIN {X 0,Y 226.222,Z 1063.447,A -85,B 0,C 180,E1 11794.817,E2 11794.817} C_VEL
LIN {X 0,Y 226.41,Z 1064.238,A -85,B 0,C 180,E1 11790.759,E2 11790.759} C_VEL
LIN {X 0,Y 226.303,Z 1063.872,A -85,B 0,C 180,E1 11786.454,E2 11786.454} C_VEL
LIN {X 0,Y 225.95,Z 1062.005,A -85,B 0,C 180,E1 11781.859,E2 11781.859} C_VEL
LIN {X 0,Y 225.754,Z 1059.052,A -85,B 0,C 180,E1 11777.466,E2 11777.466} C_VEL
LIN {X 0,Y 226.082,Z 1054.156,A -85,B 0,C 180,E1 11772.232,E2 11772.232} C_VEL
LIN {X 0,Y 227.542,Z 1047.117,A -85,B 0,C 180,E1 11766.704,E2 11766.704} C_VEL
LIN {X 0,Y 230.548,Z 1037.863,A -85,B 0,C 180,E1 11760.939,E2 11760.939} C_VEL
LIN {X 0,Y 234.919,Z 1027.327,A -85,B 0,C 180,E1 11755.658,E2 11755.658} C_VEL
LIN {X 0,Y 240.544,Z 1015.408,A -85,B 0,C 180,E1 11750.816,E2 11750.816} C_VEL
LIN {X 0,Y 247.435,Z 1001.955,A -85,B 0,C 180,E1 11746.291,E2 11746.291} C_VEL
LIN {X 0,Y 255.199,Z 987.14,A -85,B 0,C 180,E1 11742.226,E2 11742.226} C_VEL
LIN {X 0,Y 263.888,Z 970.548,A -85,B 0,C 180,E1 11738.511,E2 11738.511} C_VEL
LIN {X 0,Y 272.735,Z 953.247,A -85,B 0,C 180,E1 11735.343,E2 11735.343} C_VEL
LIN {X 0,Y 281.453,Z 935.109,A -85,B 0,C 180,E1 11732.654,E2 11732.654} C_VEL
LIN {X 0,Y 290.451,Z 914.883,A -85,B 0,C 180,E1 11730.225,E2 11730.225} C_VEL
LIN {X 0,Y 298.627,Z 894.791,A -85,B 0,C 180,E1 11728.288,E2 11728.288} C_VEL
LIN {X 0,Y 306,Z 874.24,A -85,B 0,C 180,E1 11726.716,E2 11726.716} C_VEL
LIN {X 0,Y 312.907,Z 851.921,A -85,B 0,C 180,E1 11725.377,E2 11725.377} C_VEL
LIN {X 0,Y 318.714,Z 829.607,A -85,B 0,C 180,E1 11724.362,E2 11724.362} C_VEL
LIN {X 0,Y 323.226,Z 806.974,A -85,B 0,C 180,E1 11723.578,E2 11723.578} C_VEL
LIN {X 0,Y 326.351,Z 783.594,A -85,B 0,C 180,E1 11722.948,E2 11722.948} C_VEL
LIN {X 0,Y 342.62,Z 592.286,A -85,B 0,C 180,E1 11718.87,E2 11718.87} C_VEL
LIN {X 0,Y 344.545,Z 568.752,A -85,B 0,C 180,E1 11718.352,E2 11718.352} C_VEL
LIN {X 0,Y 338.978,Z 558.566,A -85,B 0,C 180,E1 11715.526,E2 11715.526} C_VEL
LIN {X 0,Y 333.501,Z 549.403,A -85,B 0,C 180,E1 11712.29,E2 11712.29} C_VEL
LIN {X 0,Y 329.154,Z 542.4,A -85,B 0,C 180,E1 11709.176,E2 11709.176} C_VEL
LIN {X 0,Y 326.221,Z 537.927,A -85,B 0,C 180,E1 11706.599,E2 11706.599} C_VEL
LIN {X 0,Y 323.754,Z 534.188,A -85,B 0,C 180,E1 11703.895,E2 11703.895} C_VEL
LIN {X 0,Y 320.899,Z 529.63,A -85,B 0,C 180,E1 11698.928,E2 11698.928} C_VEL
LIN {X 0,Y 319.982,Z 529.037,A -85,B 0,C 180,E1 11693.721,E2 11693.721} C_VEL
LIN {X 0,Y 320.553,Z 529.71,A -85,B 0,C 180,E1 11690.665,E2 11690.665} C_VEL
LIN {X 0,Y 323.213,Z 534.512,A -85,B 0,C 180,E1 11685.488,E2 11685.488} C_VEL
LIN {X 0,Y 325.827,Z 538.799,A -85,B 0,C 180,E1 11682.498,E2 11682.498} C_VEL
LIN {X 0,Y 328.939,Z 544.004,A -85,B 0,C 180,E1 11679.725,E2 11679.725} C_VEL
LIN {X 0,Y 333.004,Z 550.882,A -85,B 0,C 180,E1 11676.791,E2 11676.791} C_VEL
LIN {X 0,Y 338.134,Z 560.061,A -85,B 0,C 180,E1 11673.716,E2 11673.716} C_VEL
LIN {X 0,Y 341.676,Z 566.925,A -85,B 0,C 180,E1 11671.853,E2 11671.853} C_VEL
LIN {X 0,Y 327.033,Z 761.371,A -85,B 0,C 180,E1 11668.07,E2 11668.07} C_VEL
LIN {X 0,Y 324.327,Z 782.467,A -85,B 0,C 180,E1 11667.405,E2 11667.405} C_VEL
LIN {X 0,Y 320.266,Z 804.074,A -85,B 0,C 180,E1 11666.467,E2 11666.467} C_VEL
LIN {X 0,Y 315.415,Z 823.781,A -85,B 0,C 180,E1 11665.348,E2 11665.348} C_VEL
LIN {X 0,Y 309.687,Z 842.279,A -85,B 0,C 180,E1 11664.012,E2 11664.012} C_VEL
LIN {X 0,Y 302.683,Z 861.342,A -85,B 0,C 180,E1 11662.293,E2 11662.293} C_VEL
LIN {X 0,Y 295.337,Z 878.579,A -85,B 0,C 180,E1 11660.372,E2 11660.372} C_VEL
LIN {X 0,Y 287.381,Z 894.925,A -85,B 0,C 180,E1 11658.121,E2 11658.121} C_VEL
LIN {X 0,Y 279.533,Z 909.317,A -85,B 0,C 180,E1 11655.675,E2 11655.675} C_VEL
LIN {X 0,Y 271.109,Z 923.45,A -85,B 0,C 180,E1 11652.735,E2 11652.735} C_VEL
LIN {X 0,Y 262.882,Z 936.179,A -85,B 0,C 180,E1 11649.434,E2 11649.434} C_VEL
LIN {X 0,Y 255.019,Z 947.467,A -85,B 0,C 180,E1 11645.746,E2 11645.746} C_VEL
LIN {X 0,Y 247.415,Z 957.908,A -85,B 0,C 180,E1 11641.421,E2 11641.421} C_VEL
LIN {X 0,Y 241.076,Z 966.41,A -85,B 0,C 180,E1 11636.877,E2 11636.877} C_VEL
LIN {X 0,Y 235.815,Z 973.448,A -85,B 0,C 180,E1 11631.908,E2 11631.908} C_VEL
LIN {X 0,Y 231.93,Z 978.701,A -85,B 0,C 180,E1 11626.789,E2 11626.789} C_VEL
LIN {X 0,Y 229.313,Z 982.556,A -85,B 0,C 180,E1 11621.316,E2 11621.316} C_VEL
LIN {X 0,Y 227.955,Z 984.803,A -85,B 0,C 180,E1 11616.043,E2 11616.043} C_VEL
LIN {X 0,Y 227.471,Z 985.627,A -85,B 0,C 180,E1 11610.756,E2 11610.756} C_VEL
LIN {X 0,Y 227.746,Z 985.112,A -85,B 0,C 180,E1 11605.215,E2 11605.215} C_VEL
LIN {X 0,Y 228.957,Z 983.167,A -85,B 0,C 180,E1 11599.686,E2 11599.686} C_VEL
LIN {X 0,Y 231.315,Z 979.688,A -85,B 0,C 180,E1 11594.198,E2 11594.198} C_VEL
LIN {X 0,Y 235.118,Z 974.421,A -85,B 0,C 180,E1 11588.809,E2 11588.809} C_VEL
